DATA_BLOCK "DB59_USV_ModTCP_RCV"
{ S7_Optimized_Access := 'FALSE' }
VERSION : 0.1
NON_RETAIN
   STRUCT
      Data : Array[0..255] of Byte;
   END_STRUCT;


BEGIN

END_DATA_BLOCK

DATA_BLOCK "DB60_USV_ModTCP_SEND"
{ S7_Optimized_Access := 'FALSE' }
VERSION : 0.1
NON_RETAIN
   STRUCT
      Data : Array[0..31] of Byte;
   END_STRUCT;


BEGIN

END_DATA_BLOCK

DATA_BLOCK "DB61_USV_ModTCP_WorkData"
{ S7_Optimized_Access := 'FALSE' }
VERSION : 0.1
   STRUCT
      REQCNT : Int;
      REQ : Array[1..10] of "T_MODBUSTCP_USV_REQ";
      REQ01 : Struct   // binär
         Reg000_l : Word;   // System - UPSStatus_BF
         Reg000_h : Word;   // System - UPSStatus_BF
         Reg002 : Int;   // System - UPSStatusChangeCause_EN
         Reg003 : DWord;   // System - MOG.OutletStatus_BF
         Reg005 : Int;   // System - Reserved []
         Reg006 : DWord;   // System - SOG[0].OutletStatus_BF
         Reg008 : Int;   // System - Reserved []
         Reg009 : DWord;   // System - SOG[1].OutletStatus_BF
         Reg011 : Int;   // System - Reserved []
         Reg012 : DWord;   // System - SOG[2].OutletStatus_BF [Bitfeld]
         Reg014 : Int;   // System - Reserved []
         Reg015 : Int;   // System - Reserved []
         Reg016 : Int;   // System - Reserved []
         Reg017 : Int;   // System - Reserved []
         Reg018 : Word;   // System - SimpleSignalingStatus_BF
         Reg019 : Word;   // System - GeneralError_BF
         Reg020 : DWord;   // System - PowerSystemError_BF [Bitfeld]
         Reg022 : Word;   // System - BatterySystemError_BF
         Reg023 : Word;   // System - ReplaceBatteryTestStatus_BF
         Reg024 : Word;   // System - RunTimeCalibrationStatus_BF
         Reg025 : Word;   // System - Battery.LifeTimeStatus_BF
         Reg026 : Word;   // System - UserInterfaceStatus_BF
      END_STRUCT;
      REQ02 : Struct   // analog
         Reg128 : DInt;   // System - RunTimeRemaining [s]
         Reg130 : Int;   // System - StateOfCharge_Pct [%]
         Reg131 : Int;   // System - Battery.Positive.VoltageDC [V]
         Reg132 : Int;   // System - Battery.Negative.VoltageDC [V]
         Reg133 : Int;   // System - Battery.Date []
         Reg134 : Int;   // System - Reserved []
         Reg135 : Int;   // System - Battery.Temperature [°C]
         Reg136 : Int;   // System - Output[0].RealPower_Pct [%]
         Reg137 : Int;   // System - Output[1].RealPower_Pct [%]
         Reg138 : Int;   // System - Output[0].ApparentPower_Pct [%]
         Reg139 : Int;   // System - Output[1].ApparentPower_Pct [%]
         Reg140 : Int;   // System - Output[0].CurrentAC [A]
         Reg141 : Int;   // System - Output[1].CurrentAC [A]
         Reg142 : Int;   // System - Output[0].VoltageAC [V]
         Reg143 : Int;   // System - Output[1].VoltageAC [V]
         Reg144 : Int;   // System - Output.Frequency [Hz]
         Reg145 : DInt;   // System - Output.Energy [Wh]
         Reg147 : Int;   // System - Bypass.InputStatus_BF [Bitfeld]
         Reg148 : Int;   // System - Bypass.VoltageAC [V]
         Reg149 : Int;   // System - Bypass.Frequency [Hz]
         Reg150 : Int;   // System - Input.InputStatus_BF [Bitfeld]
         Reg151 : Int;   // System - Input[0].VoltageAC [V]
         Reg152 : Int;   // System - Input[1].VoltageAC [V]
         Reg153 : Int;   // System - Input[2].VoltageAC [V]
         Reg154 : Int;   // System - Efficiency_EN [enum]
         Reg155 : Int;   // System - MOG.TurnOffCountdown_EN [enum]
         Reg156 : Int;   // System - MOG.TurnOnCountdown_EN [enum]
         Reg157 : DInt;   // System - MOG.StayOffCountdown_EN [enum]
         Reg159 : Int;   // System - SOG[0].TurnOffCountdown_EN [enum]
         Reg160 : Int;   // System - SOG[0].TurnOnCountdown_EN [enum]
         Reg161 : DInt;   // System - SOG[0].StayOffCountdown_EN [enum]
         Reg163 : Int;   // System - SOG[1].TurnOffCountdown_EN [enum]
         Reg164 : Int;   // System - SOG[1].TurnOnCountdown_EN [enum]
         Reg165 : DInt;   // System - SOG[1].StayOffCountdown_EN [enum]
         Reg167 : Int;   // System - SOG[2].TurnOffCountdown_EN [enum]
         Reg168 : Int;   // System - SOG[2].TurnOnCountdown_EN [enum]
         Reg169 : DInt;   // System - SOG[2].StayOffCountdown_EN [enum]
      END_STRUCT;
   END_STRUCT;


BEGIN
   REQCNT := 2;
   REQ[1].TransactID := 1;
   REQ[1].UnitID := 1;
   REQ[1].FunctionCode := 3;
   REQ[1].RegisterCount := 27;
   REQ[1].SourceDB_Num := 61;
   REQ[1].SourceDB_ByteAdr := 182;
   REQ[1].SwapBytes := TRUE;
   REQ[2].TransactID := 2;
   REQ[2].UnitID := 1;
   REQ[2].FunctionCode := 3;
   REQ[2].RegisterAdr := 128;
   REQ[2].RegisterCount := 43;
   REQ[2].SourceDB_Num := 61;
   REQ[2].SourceDB_ByteAdr := 236;

END_DATA_BLOCK

DATA_BLOCK "DB_IEC_ASDUAdr"
{ S7_Optimized_Access := 'FALSE' }
AUTHOR : SIE_GST
FAMILY : S7_IEC
NAME : P_ASDUs
VERSION : 1.6
   STRUCT
      DB_Manag { ExternalVisible := 'False'} : Struct
         Pos_of_DB { ExternalVisible := 'False'} : Byte;   // reserved for future - do not change !
         No_of_all_DBs { ExternalVisible := 'False'} : Byte;   // reserved for future - do not change !
         DB_No_Act { ExternalVisible := 'False'} : Word;   // reserved for future - do not change !
         DB_No_Prev { ExternalVisible := 'False'} : Word;   // reserved for future - do not change !
         DB_No_Next { ExternalVisible := 'False'} : Word;   // reserved for future - do not change !
         Reserved { ExternalVisible := 'False'} : Word;
      END_STRUCT;
      Info_Manag { ExternalVisible := 'False'} : Struct
         P_Byte_First_Info { ExternalVisible := 'False'} : Int;   // (Byte-) Position of first Para-Block - do not change !
         No_of_Infos { ExternalVisible := 'False'} : Int;   // 0:unspecified (DB is filled up to the end); otherwise size n of ARRAY [1..n]
         Len_Info { ExternalVisible := 'False'} : USInt;   // Difference in [byte] between two Para-Blocks - do not change !
         Len_Sort_Key { ExternalVisible := 'False'} : USInt;   // 0: without sorting; >0: Data sets are sorted ascending with x bytes
         Re_internal_usage { ExternalVisible := 'False'} : DWord;
      END_STRUCT;
      Global { ExternalVisible := 'False'} : Struct
         Glob_R1 { ExternalVisible := 'False'} : Int;
         Glob_R2 { ExternalVisible := 'False'} : Word;
      END_STRUCT;
      ASDU_Adr_Para { ExternalVisible := 'False'} : Array[0..15] of Struct
         ASDU_Address { ExternalVisible := 'False'} : DInt;   // Parameter: ASDU address
         Link_Para_DB { ExternalVisible := 'False'} : Int;   // Parameter: associated link db no / 0 -> direct (no link db available)
         Link_Para_Pos { ExternalVisible := 'False'} : Int;   // Parameter: parablock no in link db
         Error { ExternalVisible := 'False'} : Bool;   // internal
         Res_1 { ExternalVisible := 'False'} : Byte;   // internal
         Res_2 { ExternalVisible := 'False'} : DInt;   // internal
         Res_3 { ExternalVisible := 'False'} : Int;   // internal
      END_STRUCT;
   END_STRUCT;


BEGIN
   Info_Manag.P_Byte_First_Info := 24;
   Info_Manag.Len_Info := 16;
   ASDU_Adr_Para[0].ASDU_Address := DINT#25602;
   ASDU_Adr_Para[1].ASDU_Address := DINT#25860;
   ASDU_Adr_Para[2].ASDU_Address := DINT#26116;
   ASDU_Adr_Para[3].ASDU_Address := DINT#26372;
   ASDU_Adr_Para[4].ASDU_Address := DINT#26628;
   ASDU_Adr_Para[5].ASDU_Address := DINT#26884;
   ASDU_Adr_Para[6].ASDU_Address := DINT#27140;
   ASDU_Adr_Para[7].ASDU_Address := DINT#27396;
   ASDU_Adr_Para[8].ASDU_Address := DINT#27652;
   ASDU_Adr_Para[9].ASDU_Address := DINT#28164;
   ASDU_Adr_Para[10].ASDU_Address := DINT#28420;
   ASDU_Adr_Para[11].ASDU_Address := DINT#28676;
   ASDU_Adr_Para[12].ASDU_Address := DINT#28932;
   ASDU_Adr_Para[13].ASDU_Address := DINT#29188;
   ASDU_Adr_Para[14].ASDU_Address := DINT#30468;
   ASDU_Adr_Para[15].ASDU_Address := DINT#5126;

END_DATA_BLOCK

DATA_BLOCK "ZEN_MW"
{ S7_Optimized_Access := 'FALSE' }
VERSION : 0.1
NON_RETAIN
   STRUCT
      Zulauf_AR_DF_ZW : DInt;   // Zulauf - Pumpwerk "Alter Rechen" - Durchfluss - Zählwert
      BB1_DF_ZW : DInt;   // Becken 1 - Ablauf - Durchfluss - Zählwert
      BB2_DF_ZW : DInt;   // Becken 2 - Ablauf - Durchfluss - Zählwert
      Zulauf_DF_ZW : DInt;   // Zulauf - Rechen - Durchfluss - Zählwert
      BB_UeSS_DF_ZW : Real;   // Becken 1+2 - Ablauf ÜSS - Durchfluss - Zählwert
      Ablauf_DF_ZW : DInt;   // Ablauf - Durchfluss - Zählwert
      Schlamm_Besch_DF_ZW : DInt;   // Schlamm - Beschickung - Durchfluss - Zählwert
      Truebwasser_DF_ZW : DInt;   // Trübwasserpumpwerk - Durchfluss - Zählwert
      BB_Biocos_DF_ZW : DInt;   // Becken 1+2 - Schlammmenge Biocos - Zählwert
      Zulauf_AR_DF_ZW_Tag : DInt;   // Zulauf - Pumpwerk "Alter Rechen" - Durchfluss - Zählwert Tag
      BB1_DF_ZW_Tag : DInt;   // Becken 1 - Ablauf - Durchfluss - Zählwert Tag
      BB2_DF_ZW_Tag : DInt;   // Becken 2 - Ablauf - Durchfluss - Zählwert Tag
      Zulauf_DF_ZW_Tag : DInt;   // Zulauf - Rechen - Durchfluss - Zählwert Tag
      BB_UeSS_DF_ZW_Tag : Real;   // Becken 1+2 - Ablauf ÜSS - Durchfluss - Zählwert Tag
      Ablauf_DF_ZW_Tag : DInt;   // Ablauf - Durchfluss - Zählwert Tag
      Schlamm_Besch_DF_ZW_Tag : DInt;   // Schlamm - Beschickung - Durchfluss - Zählwert Tag
      Truebwasser_DF_ZW_Tag : DInt;   // Trübwasserpumpwerk - Durchfluss - Zählwert Tag
      BB_Biocos_DF_ZW_Tag : DInt;   // Becken 1+2 - Schlammmenge Biocos - Zählwert Tag
      Zulauf_AR_DF_ZW_Vortag : DInt;   // Zulauf - Pumpwerk "Alter Rechen" - Durchfluss - Zählwert Vortag
      BB1_DF_ZW_Vortag : DInt;   // Becken 1 - Ablauf - Durchfluss - Zählwert Vortag
      BB2_DF_ZW_Vortag : DInt;   // Becken 2 - Ablauf - Durchfluss - Zählwert Vortag
      Zulauf_DF_ZW_Vortag : DInt;   // Zulauf - Rechen - Durchfluss - Zählwert Vortag
      BB_UeSS_DF_ZW_Vortag : Real;   // Becken 1+2 - Ablauf ÜSS - Durchfluss - Zählwert Vortag
      Ablauf_DF_ZW_Vortag : DInt;   // Ablauf - Durchfluss - Zählwert Vortag
      Schlamm_Besch_DF_ZW_Vortag : DInt;   // Schlamm - Beschickung - Durchfluss - Zählwert Vortag
      Truebwasser_DF_ZW_Vortag : DInt;   // Trübwasserpumpwerk - Durchfluss - Zählwert Vortag
      BB_Biocos_DF_ZW_Vortag : DInt;   // Becken 1+2 - Schlammmenge Biocos - Zählwert Vortag
      ZEN_Bed_ID : DInt;   // UV BG Bedienstelle - Bediener aktuell - ID
      ZEN_ESK_Stufe_act : DInt;   // UV BG - Einschaltkaskade - aktive Schaltpriorität
      ZEN_ESK_NLZ_Stufe_req : DInt;   // UV BG - Einschaltkaskade - Nachlaufzeit max. für angeforderte Schaltpriorität
      ZEN_ESK_Stufe_req : DInt;   // UV BG - Einschaltkaskade - Anforderung Schaltpriorität
      BB_Auto_GeblW_ZZ_IW : DInt;   // Steuerung Belüftung - Automatik - Zykluszeit Gebläsetausch - Istwert
      Biocos1_Auto_A_Zt_P1_SW : DInt;   // Steuerung Biocos 1 - Automatik - Sollwert A-Phase (Rechenwert U+V) - Parametersatz 1
      Biocos1_Auto_Bel_Frg_P1_SW : DInt;   // Steuerung Biocos 1 - Automatik - Sollwert Belüftungsphase Freigabe (Rechenwert V-Verz.) - Parametersatz 1
      Biocos1_Auto_A_Zt_P2_SW : DInt;   // Steuerung Biocos 1 - Automatik - Sollwert A-Phase (Rechenwert U+V) - Parametersatz 2
      Biocos1_Auto_Bel_Frg_P2_SW : DInt;   // Steuerung Biocos 1 - Automatik - Sollwert Belüftungsphase Freigabe (Rechenwert V-Verz.) - Parametersatz 2
      ZEN_Res_DB102_144_0 : DInt;   // Reserve
      Biocos1_Auto_U_Zt_Px_IW : DInt;   // Steuerung Biocos 1 - Automatik - Sollwert U-Phase - Parameter aktiv
      Biocos1_Auto_V_Zt_Px_IW : DInt;   // Steuerung Biocos 1 - Automatik - Sollwert V-Phase - Parameter aktiv
      Biocos1_Auto_A_Zt_Px_IW : DInt;   // Steuerung Biocos 1 - Automatik - Sollwert A-Phase (Rechenwert U+V) - Parameter aktiv
      Biocos1_Auto_Bel_Vz_Px_IW : DInt;   // Steuerung Biocos 1 - Automatik - Sollwert Verzögerungszeit Belüftungsphase - Parameter aktiv
      Biocos1_Auto_Bel_Frg_Px_IW : DInt;   // Steuerung Biocos 1 - Automatik - Sollwert Belüftungsphase Freigabe (Rechenwert V-Verz.) - Parameter aktiv
      Biocos1_Auto_Bel_Int_Px_IW : DInt;   // Steuerung Biocos 1 - Automatik - Sollwert Anzahl Belüftungsintervalle - Parameter aktiv
      Biocos1_Auto_Bel_Int_Zt_Px_IW : DInt;   // Steuerung Biocos 1 - Automatik - Sollwert Belüftungsdauer (fest) pro Intervall - Parameter aktiv
      Biocos1_Auto_UeSS_Zt_Px_IW : DInt;   // Steuerung Biocos 1 - Automatik - Sollwert ÜSS-Abzug Dauer - Parameter aktiv
      Biocos1_Auto_UeSS_Df_Px_IW : Real;   // Steuerung Biocos 1 - Automatik - Sollwert ÜSS-Abzug Menge - Parameter aktiv
      Biocos1_Auto_SR1_Zt_Px_IW : DInt;   // Steuerung Biocos 1 - Automatik - Sollwert Dauer Schlammrückführung SU-Becken 1 - Parameter aktiv
      Biocos1_Auto_SR2_Zt_Px_IW : DInt;   // Steuerung Biocos 1 - Automatik - Sollwert Dauer Schlammrückführung SU-Becken 2 - Parameter aktiv
      ZEN_Res_DB102_192_0 : DInt;   // Reserve
      Biocos1_Auto_UeSS_Zyk_IW : DInt;   // Steuerung Biocos 1 - Automatik - Zyklen bis ÜSS-Abzug - Istwert
      Biocos1_Auto_U1_Zt_IW : DInt;   // Steuerung Biocos 1 - Automatik - U-Phase SU-Becken 1 - Istwert
      Biocos1_Auto_V1_Zt_IW : DInt;   // Steuerung Biocos 1 - Automatik - V-Phase SU-Becken 1 - Istwert
      Biocos1_Auto_A1_Zt_IW : DInt;   // Steuerung Biocos 1 - Automatik - A-Phase SU-Becken 1 - Istwert
      Biocos1_Auto_U2_Zt_IW : DInt;   // Steuerung Biocos 1 - Automatik - U-Phase SU-Becken 2 - Istwert
      Biocos1_Auto_V2_Zt_IW : DInt;   // Steuerung Biocos 1 - Automatik - V-Phase SU-Becken 2 - Istwert
      Biocos1_Auto_A2_Zt_IW : DInt;   // Steuerung Biocos 1 - Automatik - A-Phase SU-Becken 2 - Istwert
      Biocos1_Auto_Bel_Vz_IW : DInt;   // Steuerung Biocos 1 - Automatik - Verzögerungszeit Belüftungsphase - Istwert
      Biocos1_Auto_Bel_Frg_IW : DInt;   // Steuerung Biocos 1 - Automatik - Belüftungsphase - Istwert
      Biocos1_Auto_Bel_Int_IW : DInt;   // Steuerung Biocos 1 - Automatik - Belüftungsintervall - Istwert
      Biocos1_Auto_Bel_Int_Zt_IW : DInt;   // Steuerung Biocos 1 - Automatik - Belüftungsdauer im Intervall - Istwert
      Biocos1_Auto_UeSS_Zt_IW : DInt;   // Steuerung Biocos 1 - Automatik - ÜSS-Abzug Dauer - Istwert
      Biocos1_Auto_UeSS_Df_IW : Real;   // Steuerung Biocos 1 - Automatik - ÜSS-Abzug Menge - Istwert
      Biocos1_Auto_SR1_Zt_IW : DInt;   // Steuerung Biocos 1 - Automatik - Schlammrückführung SU-Becken 1 - Istwert
      Biocos1_Auto_SR2_Zt_IW : DInt;   // Steuerung Biocos 1 - Automatik - Schlammrückführung SU-Becken 2 - Istwert
      ZEN_Res_DB102_256_0 : DInt;   // Reserve
      Biocos2_Auto_A_Zt_P1_SW : DInt;   // Steuerung Biocos 2 - Automatik - Sollwert A-Phase (Rechenwert U+V) - Parametersatz 1
      Biocos2_Auto_Bel_Frg_P1_SW : DInt;   // Steuerung Biocos 2 - Automatik - Sollwert Belüftungsphase Freigabe (Rechenwert V-Verz.) - Parametersatz 1
      Biocos2_Auto_A_Zt_P2_SW : DInt;   // Steuerung Biocos 2 - Automatik - Sollwert A-Phase (Rechenwert U+V) - Parametersatz 2
      Biocos2_Auto_Bel_Frg_P2_SW : DInt;   // Steuerung Biocos 2 - Automatik - Sollwert Belüftungsphase Freigabe (Rechenwert V-Verz.) - Parametersatz 2
      ZEN_Res_DB102_276_0 : DInt;   // Reserve
      Biocos2_Auto_U_Zt_Px_IW : DInt;   // Steuerung Biocos 2 - Automatik - Sollwert U-Phase - Parameter aktiv
      Biocos2_Auto_V_Zt_Px_IW : DInt;   // Steuerung Biocos 2 - Automatik - Sollwert V-Phase - Parameter aktiv
      Biocos2_Auto_A_Zt_Px_IW : DInt;   // Steuerung Biocos 2 - Automatik - Sollwert A-Phase (Rechenwert U+V) - Parameter aktiv
      Biocos2_Auto_Bel_Vz_Px_IW : DInt;   // Steuerung Biocos 2 - Automatik - Sollwert Verzögerungszeit Belüftungsphase - Parameter aktiv
      Biocos2_Auto_Bel_Frg_Px_IW : DInt;   // Steuerung Biocos 2 - Automatik - Sollwert Belüftungsphase Freigabe (Rechenwert V-Verz.) - Parameter aktiv
      Biocos2_Auto_Bel_Int_Px_IW : DInt;   // Steuerung Biocos 2 - Automatik - Sollwert Anzahl Belüftungsintervalle - Parameter aktiv
      Biocos2_Auto_Bel_Int_Zt_Px_IW : DInt;   // Steuerung Biocos 2 - Automatik - Sollwert Belüftungsdauer (fest) pro Intervall - Parameter aktiv
      Biocos2_Auto_UeSS_Zt_Px_IW : DInt;   // Steuerung Biocos 2 - Automatik - Sollwert ÜSS-Abzug Dauer - Parameter aktiv
      Biocos2_Auto_UeSS_Df_Px_IW : Real;   // Steuerung Biocos 2 - Automatik - Sollwert ÜSS-Abzug Menge - Parameter aktiv
      Biocos2_Auto_SR1_Zt_Px_IW : DInt;   // Steuerung Biocos 2 - Automatik - Sollwert Dauer Schlammrückführung SU-Becken 1 - Parameter aktiv
      Biocos2_Auto_SR2_Zt_Px_IW : DInt;   // Steuerung Biocos 2 - Automatik - Sollwert Dauer Schlammrückführung SU-Becken 2 - Parameter aktiv
      ZEN_Res_DB102_324_0 : DInt;   // Reserve
      Biocos2_Auto_UeSS_Zyk_IW : DInt;   // Steuerung Biocos 2 - Automatik - Zyklen bis ÜSS-Abzug - Istwert
      Biocos2_Auto_U1_Zt_IW : DInt;   // Steuerung Biocos 2 - Automatik - U-Phase SU-Becken 1 - Istwert
      Biocos2_Auto_V1_Zt_IW : DInt;   // Steuerung Biocos 2 - Automatik - V-Phase SU-Becken 1 - Istwert
      Biocos2_Auto_A1_Zt_IW : DInt;   // Steuerung Biocos 2 - Automatik - A-Phase SU-Becken 1 - Istwert
      Biocos2_Auto_U2_Zt_IW : DInt;   // Steuerung Biocos 2 - Automatik - U-Phase SU-Becken 2 - Istwert
      Biocos2_Auto_V2_Zt_IW : DInt;   // Steuerung Biocos 2 - Automatik - V-Phase SU-Becken 2 - Istwert
      Biocos2_Auto_A2_Zt_IW : DInt;   // Steuerung Biocos 2 - Automatik - A-Phase SU-Becken 2 - Istwert
      Biocos2_Auto_Bel_Vz_IW : DInt;   // Steuerung Biocos 2 - Automatik - Verzögerungszeit Belüftungsphase - Istwert
      Biocos2_Auto_Bel_Frg_IW : DInt;   // Steuerung Biocos 2 - Automatik - Belüftungsphase - Istwert
      Biocos2_Auto_Bel_Int_IW : DInt;   // Steuerung Biocos 2 - Automatik - Belüftungsintervall - Istwert
      Biocos2_Auto_Bel_Int_Zt_IW : DInt;   // Steuerung Biocos 2 - Automatik - Belüftungsdauer im Intervall - Istwert
      Biocos2_Auto_UeSS_Zt_IW : DInt;   // Steuerung Biocos 2 - Automatik - ÜSS-Abzug Dauer - Istwert
      Biocos2_Auto_UeSS_Df_IW : Real;   // Steuerung Biocos 2 - Automatik - ÜSS-Abzug Menge - Istwert
      Biocos2_Auto_SR1_Zt_IW : DInt;   // Steuerung Biocos 2 - Automatik - Schlammrückführung SU-Becken 1 - Istwert
      Biocos2_Auto_SR2_Zt_IW : DInt;   // Steuerung Biocos 2 - Automatik - Schlammrückführung SU-Becken 2 - Istwert
      Schlamm_Besch_Auto_Menge_IW : DInt;   // Steuerung Beschickung Schlammbeete - Menge Beschickung - Istwert
      PO4_Elim_DosP_Status_DF_SW : Real;   // Steuerung PO4-Elimination - Status Dosierpumpe - Menge Fällmittel - Sollwert
      PO4_Elim_DosP_Status_DF_IW : Real;   // Steuerung PO4-Elimination - Status Dosierpumpe - Menge Fällmittel - Istwert
      PO4_Elim_DosP_Status_Dr_IW : Real;   // Steuerung PO4-Elimination - Status Dosierpumpe - Druck (ohne Luftdruck) - Istwert
      PO4_Elim_DosP_Status_DF_ZW : Real;   // Steuerung PO4-Elimination - Status Dosierpumpe - Menge Fällmittel - Zählwert
      Biocos1_Auto_Bel_O2_Reg_IW : Real;   // Steuerung Biocos 1 - Automatik O2-Regler - Vorgabe Automatik Blockdrehzahl für Ansteuerung Gebläse
      Biocos2_Auto_Bel_O2_Reg_IW : Real;   // Steuerung Biocos 2 - Automatik O2-Regler - Vorgabe Automatik Blockdrehzahl für Ansteuerung Gebläse
      BB_G1_KS_Druck_Netz : Real;   // Belebung - SigmaControl Gebläse 1 - Messwerte - Netzdruck
      BB_G1_KS_Temp_Verdicht : Real;   // Belebung - SigmaControl Gebläse 1 - Messwerte - Verdichtungsendtemperatur (t2)
      BB_G1_KS_Temp_Schallhaube : Real;   // Belebung - SigmaControl Gebläse 1 - Messwerte - Temperatur Schalldämmhaube (t_S)
      BB_G1_KS_Temp_Ansaug : Real;   // Belebung - SigmaControl Gebläse 1 - Messwerte - Ansaugtemperatur (t1)
      BB_G1_KS_Temp_Oel : Real;   // Belebung - SigmaControl Gebläse 1 - Messwerte - Öltemperatur (t3 )
      BB_G1_KS_Temp_Wicklung : Real;   // Belebung - SigmaControl Gebläse 1 - Messwerte - Wicklungstemperatur Hauptmotor
      BB_G1_KS_Volumenstrom : Real;   // Belebung - SigmaControl Gebläse 1 - Messwerte - Volumenstrom
      BB_G1_KS_Motorfrequenz : Real;   // Belebung - SigmaControl Gebläse 1 - Messwerte - Motorfrequenz
      BB_G1_KS_Motordrehzahl : Real;   // Belebung - SigmaControl Gebläse 1 - Messwerte - Motordrehzahl
      BB_G1_KS_Blockdrehzahl : Real;   // Belebung - SigmaControl Gebläse 1 - Messwerte - Blockdrehzahl
      BB_G2_KS_Druck_Netz : Real;   // Belebung - SigmaControl Gebläse 2 - Messwerte - Netzdruck
      BB_G2_KS_Temp_Verdicht : Real;   // Belebung - SigmaControl Gebläse 2 - Messwerte - Verdichtungsendtemperatur (t2)
      BB_G2_KS_Temp_Schallhaube : Real;   // Belebung - SigmaControl Gebläse 2 - Messwerte - Temperatur Schalldämmhaube (t_S)
      BB_G2_KS_Temp_Ansaug : Real;   // Belebung - SigmaControl Gebläse 2 - Messwerte - Ansaugtemperatur (t1)
      BB_G2_KS_Temp_Oel : Real;   // Belebung - SigmaControl Gebläse 2 - Messwerte - Öltemperatur (t3 )
      BB_G2_KS_Temp_Wicklung : Real;   // Belebung - SigmaControl Gebläse 2 - Messwerte - Wicklungstemperatur Hauptmotor
      BB_G2_KS_Volumenstrom : Real;   // Belebung - SigmaControl Gebläse 2 - Messwerte - Volumenstrom
      BB_G2_KS_Motorfrequenz : Real;   // Belebung - SigmaControl Gebläse 2 - Messwerte - Motorfrequenz
      BB_G2_KS_Motordrehzahl : Real;   // Belebung - SigmaControl Gebläse 2 - Messwerte - Motordrehzahl
      BB_G2_KS_Blockdrehzahl : Real;   // Belebung - SigmaControl Gebläse 2 - Messwerte - Blockdrehzahl
      BB_G3_KS_Druck_Netz : Real;   // Belebung - SigmaControl Gebläse 3 - Messwerte - Netzdruck
      BB_G3_KS_Temp_Verdicht : Real;   // Belebung - SigmaControl Gebläse 3 - Messwerte - Verdichtungsendtemperatur (t2)
      BB_G3_KS_Temp_Schallhaube : Real;   // Belebung - SigmaControl Gebläse 3 - Messwerte - Temperatur Schalldämmhaube (t_S)
      BB_G3_KS_Temp_Ansaug : Real;   // Belebung - SigmaControl Gebläse 3 - Messwerte - Ansaugtemperatur (t1)
      BB_G3_KS_Temp_Oel : Real;   // Belebung - SigmaControl Gebläse 3 - Messwerte - Öltemperatur (t3 )
      BB_G3_KS_Temp_Wicklung : Real;   // Belebung - SigmaControl Gebläse 3 - Messwerte - Wicklungstemperatur Hauptmotor
      BB_G3_KS_Volumenstrom : Real;   // Belebung - SigmaControl Gebläse 3 - Messwerte - Volumenstrom
      BB_G3_KS_Motorfrequenz : Real;   // Belebung - SigmaControl Gebläse 3 - Messwerte - Motorfrequenz
      BB_G3_KS_Motordrehzahl : Real;   // Belebung - SigmaControl Gebläse 3 - Messwerte - Motordrehzahl
      BB_G3_KS_Blockdrehzahl : Real;   // Belebung - SigmaControl Gebläse 3 - Messwerte - Blockdrehzahl
      Umwelt_RM_ZW : Real;   // Wetterstation - Regenmenge - Zählwert
      Umwelt_RM_ZW_Tag : Real;   // Wetterstation - Regenmenge - Zählwert Tag
      Umwelt_RM_ZW_Vortag : Real;   // Wetterstation - Regenmenge - Zählwert Vortag
      RunTimeRemaining : Real;   // USV-Anlage - Status - verbleibende Laufzeit
      StateOfCharge_Pct : Real;   // USV-Anlage - Status - Batterieladung
      RES : Array[0..9] of Byte;
   END_STRUCT;


BEGIN
   Zulauf_AR_DF_ZW := 583302;
   BB1_DF_ZW := 0;
   BB2_DF_ZW := 0;
   Zulauf_DF_ZW := 1741318;
   BB_UeSS_DF_ZW := 82177.4;
   Ablauf_DF_ZW := 1542271;
   Schlamm_Besch_DF_ZW := 53300;
   Truebwasser_DF_ZW := 207644;
   BB_Biocos_DF_ZW := 0;
   Zulauf_AR_DF_ZW_Tag := 0;
   BB1_DF_ZW_Tag := 0;
   BB2_DF_ZW_Tag := 0;
   Zulauf_DF_ZW_Tag := 1066;
   BB_UeSS_DF_ZW_Tag := 39.0;
   Ablauf_DF_ZW_Tag := 869;
   Schlamm_Besch_DF_ZW_Tag := 0;
   Truebwasser_DF_ZW_Tag := 89;
   BB_Biocos_DF_ZW_Tag := 0;
   Zulauf_AR_DF_ZW_Vortag := 0;
   BB1_DF_ZW_Vortag := 0;
   BB2_DF_ZW_Vortag := 0;
   Zulauf_DF_ZW_Vortag := 905;
   BB_UeSS_DF_ZW_Vortag := 39.0;
   Ablauf_DF_ZW_Vortag := 815;
   Schlamm_Besch_DF_ZW_Vortag := 0;
   Truebwasser_DF_ZW_Vortag := 90;
   BB_Biocos_DF_ZW_Vortag := 0;
   ZEN_Bed_ID := 0;
   ZEN_ESK_Stufe_act := 0;
   ZEN_ESK_NLZ_Stufe_req := 0;
   ZEN_ESK_Stufe_req := 0;
   BB_Auto_GeblW_ZZ_IW := 22;
   Biocos1_Auto_A_Zt_P1_SW := 60;
   Biocos1_Auto_Bel_Frg_P1_SW := 33;
   Biocos1_Auto_A_Zt_P2_SW := 90;
   Biocos1_Auto_Bel_Frg_P2_SW := 71;
   ZEN_Res_DB102_144_0 := 0;
   Biocos1_Auto_U_Zt_Px_IW := 15;
   Biocos1_Auto_V_Zt_Px_IW := 45;
   Biocos1_Auto_A_Zt_Px_IW := 60;
   Biocos1_Auto_Bel_Vz_Px_IW := 720;
   Biocos1_Auto_Bel_Frg_Px_IW := 33;
   Biocos1_Auto_Bel_Int_Px_IW := 3;
   Biocos1_Auto_Bel_Int_Zt_Px_IW := 300;
   Biocos1_Auto_UeSS_Zt_Px_IW := 8;
   Biocos1_Auto_UeSS_Df_Px_IW := 1.6;
   Biocos1_Auto_SR1_Zt_Px_IW := 3;
   Biocos1_Auto_SR2_Zt_Px_IW := 3;
   ZEN_Res_DB102_192_0 := 0;
   Biocos1_Auto_UeSS_Zyk_IW := 1;
   Biocos1_Auto_U1_Zt_IW := 15;
   Biocos1_Auto_V1_Zt_IW := 45;
   Biocos1_Auto_A1_Zt_IW := 4;
   Biocos1_Auto_U2_Zt_IW := 15;
   Biocos1_Auto_V2_Zt_IW := 4;
   Biocos1_Auto_A2_Zt_IW := 60;
   Biocos1_Auto_Bel_Vz_IW := 720;
   Biocos1_Auto_Bel_Frg_IW := 4;
   Biocos1_Auto_Bel_Int_IW := 0;
   Biocos1_Auto_Bel_Int_Zt_IW := 183;
   Biocos1_Auto_UeSS_Zt_IW := 8;
   Biocos1_Auto_UeSS_Df_IW := 1.695313;
   Biocos1_Auto_SR1_Zt_IW := 3;
   Biocos1_Auto_SR2_Zt_IW := 3;
   ZEN_Res_DB102_256_0 := 0;
   Biocos2_Auto_A_Zt_P1_SW := 60;
   Biocos2_Auto_Bel_Frg_P1_SW := 33;
   Biocos2_Auto_A_Zt_P2_SW := 90;
   Biocos2_Auto_Bel_Frg_P2_SW := 71;
   ZEN_Res_DB102_276_0 := 0;
   Biocos2_Auto_U_Zt_Px_IW := 15;
   Biocos2_Auto_V_Zt_Px_IW := 45;
   Biocos2_Auto_A_Zt_Px_IW := 60;
   Biocos2_Auto_Bel_Vz_Px_IW := 720;
   Biocos2_Auto_Bel_Frg_Px_IW := 33;
   Biocos2_Auto_Bel_Int_Px_IW := 3;
   Biocos2_Auto_Bel_Int_Zt_Px_IW := 300;
   Biocos2_Auto_UeSS_Zt_Px_IW := 8;
   Biocos2_Auto_UeSS_Df_Px_IW := 1.6;
   Biocos2_Auto_SR1_Zt_Px_IW := 3;
   Biocos2_Auto_SR2_Zt_Px_IW := 3;
   ZEN_Res_DB102_324_0 := 0;
   Biocos2_Auto_UeSS_Zyk_IW := 0;
   Biocos2_Auto_U1_Zt_IW := 15;
   Biocos2_Auto_V1_Zt_IW := 4;
   Biocos2_Auto_A1_Zt_IW := 60;
   Biocos2_Auto_U2_Zt_IW := 15;
   Biocos2_Auto_V2_Zt_IW := 45;
   Biocos2_Auto_A2_Zt_IW := 4;
   Biocos2_Auto_Bel_Vz_IW := 720;
   Biocos2_Auto_Bel_Frg_IW := 4;
   Biocos2_Auto_Bel_Int_IW := 0;
   Biocos2_Auto_Bel_Int_Zt_IW := 217;
   Biocos2_Auto_UeSS_Zt_IW := 8;
   Biocos2_Auto_UeSS_Df_IW := 1.601563;
   Biocos2_Auto_SR1_Zt_IW := 3;
   Biocos2_Auto_SR2_Zt_IW := 3;
   Schlamm_Besch_Auto_Menge_IW := 50;
   PO4_Elim_DosP_Status_DF_SW := 0.2077;
   PO4_Elim_DosP_Status_DF_IW := 0.2053;
   PO4_Elim_DosP_Status_Dr_IW := 1.0;
   PO4_Elim_DosP_Status_DF_ZW := 34901.2;
   Biocos1_Auto_Bel_O2_Reg_IW := 3000.0;
   Biocos2_Auto_Bel_O2_Reg_IW := 3000.0;
   BB_G1_KS_Druck_Netz := 576.0;
   BB_G1_KS_Temp_Verdicht := 63.9;
   BB_G1_KS_Temp_Schallhaube := -3276.8;
   BB_G1_KS_Temp_Ansaug := 20.7;
   BB_G1_KS_Temp_Oel := 37.5;
   BB_G1_KS_Temp_Wicklung := 45.6;
   BB_G1_KS_Volumenstrom := 294.0;
   BB_G1_KS_Motorfrequenz := 17.0;
   BB_G1_KS_Motordrehzahl := 1055.0;
   BB_G1_KS_Blockdrehzahl := 2997.0;
   BB_G2_KS_Druck_Netz := 565.0;
   BB_G2_KS_Temp_Verdicht := 63.9;
   BB_G2_KS_Temp_Schallhaube := -3276.8;
   BB_G2_KS_Temp_Ansaug := 20.7;
   BB_G2_KS_Temp_Oel := 35.5;
   BB_G2_KS_Temp_Wicklung := 44.1;
   BB_G2_KS_Volumenstrom := 300.0;
   BB_G2_KS_Motorfrequenz := 17.0;
   BB_G2_KS_Motordrehzahl := 1057.0;
   BB_G2_KS_Blockdrehzahl := 3003.0;
   BB_G3_KS_Druck_Netz := 0.0;
   BB_G3_KS_Temp_Verdicht := 18.8;
   BB_G3_KS_Temp_Schallhaube := -3276.8;
   BB_G3_KS_Temp_Ansaug := 18.6;
   BB_G3_KS_Temp_Oel := 18.7;
   BB_G3_KS_Temp_Wicklung := 18.3;
   BB_G3_KS_Volumenstrom := 0.0;
   BB_G3_KS_Motorfrequenz := 0.0;
   BB_G3_KS_Motordrehzahl := 0.0;
   BB_G3_KS_Blockdrehzahl := 0.0;
   RES[0] := 16#00;
   RES[1] := 16#00;
   RES[2] := 16#00;
   RES[3] := 16#00;
   RES[4] := 16#00;
   RES[5] := 16#00;
   RES[6] := 16#00;
   RES[7] := 16#00;
   RES[8] := 16#00;
   RES[9] := 16#00;

END_DATA_BLOCK

DATA_BLOCK "ZEN_Meld"
{ S7_Optimized_Access := 'FALSE' }
VERSION : 0.1
   STRUCT
      E_Zulauf_AR_P1_Ein : Bool;   // Zulauf - Pumpwerk "Alter Rechen" - Pumpe 1 - Betrieb
      E_Zulauf_AR_P1_St : Bool;   // Zulauf - Pumpwerk "Alter Rechen" - Pumpe 1 - Störung
      E_Zulauf_AR_SS : Bool;   // Zulauf - Pumpwerk "Alter Rechen" - Sammelstörung
      E_Zulauf_AR_P2_Ein : Bool;   // Zulauf - Pumpwerk "Alter Rechen" - Pumpe 2 - Betrieb
      E_Zulauf_AR_P2_St : Bool;   // Zulauf - Pumpwerk "Alter Rechen" - Pumpe 2 - Störung
      E_Zulauf_AR_HW : Bool;   // Zulauf - Pumpwerk "Alter Rechen" - Hochwasser
      E_Zulauf_AR_Niv_St : Bool;   // Zulauf - Pumpwerk "Alter Rechen" - Niveau - Störung
      E_Zulauf_AR_DF_ZI : Bool;   // Zulauf - Pumpwerk "Alter Rechen" - Durchfluss - Impuls
      E_Zulauf_AR_DF_St : Bool;   // Zulauf - Pumpwerk "Alter Rechen" - Durchfluss - Störung
      E_Ablauf_pH_St : Bool;   // Ablauf - pH-Wert - Störung
      E_Ablauf_O2_St : Bool;   // Ablauf - O2-Gehalt - Störung
      E_Ablauf_DF_ZI : Bool;   // Ablauf - Durchfluss - Impuls
      E_Ablauf_DF_St : Bool;   // Ablauf - Durchfluss - Störung
      E_BB_UeSS_DF_ZI : Bool;   // Becken 1+2 - Ablauf ÜSS - Durchfluss - Impuls
      E_ZEN_Res_1_6 : Bool;   // Reserve
      E_ZEN_Res_1_7 : Bool;   // Reserve
      E_NSHV_SS1_St : Bool;   // NSHV Steuerspannungsüberwachung 1 - Störung
      E_NSHV_SS2_St : Bool;   // NSHV Steuerspannungsüberwachung 2 - Störung
      E_NSHV_N02_AF_St : Bool;   // NSHV Sicherungsüberwachung Feld N02 - Störung
      E_NSHV_N03_AF_St : Bool;   // NSHV Sicherungsüberwachung Feld N03 - Störung
      E_NSHV_N04_AF_St : Bool;   // NSHV Sicherungsüberwachung Feld N04 - Störung
      E_NSHV_LS_Aus : Bool;   // NSHV Netzleistungsschalter - Aus
      E_NSHV_LS_St : Bool;   // NSHV Netzleistungsschalter - ausgelöst
      E_NSHV_NA : Bool;   // NSHV Netzspannungsüberwachung - ausgelöst
      E_ZEN_Res_3_0 : Bool;   // Reserve
      E_ZEN_Res_3_1 : Bool;   // Reserve
      E_ZEN_Res_3_2 : Bool;   // Reserve
      E_ZEN_Res_3_3 : Bool;   // Reserve
      E_ZEN_Res_3_4 : Bool;   // Reserve
      E_ZEN_Res_3_5 : Bool;   // Reserve
      E_ZEN_Res_3_6 : Bool;   // Reserve
      E_ZEN_Res_3_7 : Bool;   // Reserve
      E_BB_G1_Ein : Bool;   // Belebung - Gebläse 1 - Betrieb
      E_BB_G1_St : Bool;   // Belebung - Gebläse 1 - Störung
      E_BB_G1_Bed_vOrt : Bool;   // Belebung - Gebläse 1 - vor-Ort-Hand
      E_BB_G1_Bed_Fern : Bool;   // Belebung - Gebläse 1 - vor-Ort-Fern
      E_BB_G1_AF_St : Bool;   // Belebung - Gebläse 1 - Steuersicherung ausgelöst
      E_BB_SHL_G1_Ein : Bool;   // Belebung - Schallhaubenlüfter Gebläse 1 - Betrieb
      E_BB_SHL_G1_St : Bool;   // Belebung - Schallhaubenlüfter Gebläse 1 - Störung
      E_BB_G2_Ein : Bool;   // Belebung - Gebläse 2 - Betrieb
      E_BB_G2_St : Bool;   // Belebung - Gebläse 2 - Störung
      E_BB_G2_Bed_vOrt : Bool;   // Belebung - Gebläse 2 - vor-Ort-Hand
      E_BB_G2_Bed_Fern : Bool;   // Belebung - Gebläse 2 - vor-Ort-Fern
      E_BB_G2_AF_St : Bool;   // Belebung - Gebläse 2 - Steuersicherung ausgelöst
      E_BB_SHL_G2_Ein : Bool;   // Belebung - Schallhaubenlüfter Gebläse 2 - Betrieb
      E_BB_SHL_G2_St : Bool;   // Belebung - Schallhaubenlüfter Gebläse 2 - Störung
      E_BB_G3_Ein : Bool;   // Belebung - Gebläse 3 - Betrieb
      E_BB_G3_St : Bool;   // Belebung - Gebläse 3 - Störung
      E_BB_G3_Bed_vOrt : Bool;   // Belebung - Gebläse 3 - vor-Ort-Hand
      E_BB_G3_Bed_Fern : Bool;   // Belebung - Gebläse 3 - vor-Ort-Fern
      E_BB_G3_AF_St : Bool;   // Belebung - Gebläse 3 - Steuersicherung ausgelöst
      E_BB_SHL_G3_Ein : Bool;   // Belebung - Schallhaubenlüfter Gebläse 3 - Betrieb
      E_BB_SHL_G3_St : Bool;   // Belebung - Schallhaubenlüfter Gebläse 3 - Störung
      E_BB_AV_Ein : Bool;   // Belebung - Gebläsestation - Abluftventilator - Betrieb
      E_BB_AV_St : Bool;   // Belebung - Gebläsestation - Abluftventilator - Störung
      E_BB_AV_AF_St : Bool;   // Belebung - Gebläsestation - Abluftventilator - Steuersicherung ausgelöst
      E_BB_RT : Bool;   // Belebung - Gebläsestation - Raumthermostat - Grenztemperatur erreicht
      E_BB1_SR_K_Ein : Bool;   // Becken 1 - Druckluftkompressor Schlammrückführung
      E_BB1_SR_K_St : Bool;   // Becken 1 - Druckluftkompressor Schlammrückführung
      E_BB1_SR_K_AF_St : Bool;   // Becken 1 - Druckluftkompressor Schlammrückführung
      E_BB_LS1_EA : Bool;   // Belebung - Gebläsestation - Luftwegschieber 1 - Endlage Auf
      E_BB_LS1_EZ : Bool;   // Belebung - Gebläsestation - Luftwegschieber 1 - Endlage Zu
      E_BB_LS1_St : Bool;   // Belebung - Gebläsestation - Luftwegschieber 1 - Störung
      E_BB_LS1_Bed_vOrt : Bool;   // Belebung - Gebläsestation - Luftwegschieber 1 - vor-Ort-Hand
      E_BB_LS1_Bed_Fern : Bool;   // Belebung - Gebläsestation - Luftwegschieber 1 - vor-Ort-Fern
      E_BB_LS1_AF_St : Bool;   // Belebung - Gebläsestation - Luftwegschieber 1 - Steuersicherung ausgelöst
      E_BB_LS2_EA : Bool;   // Belebung - Gebläsestation - Luftwegschieber 2 - Endlage Auf
      E_BB_LS2_EZ : Bool;   // Belebung - Gebläsestation - Luftwegschieber 2 - Endlage Zu
      E_BB_LS2_St : Bool;   // Belebung - Gebläsestation - Luftwegschieber 2 - Störung
      E_BB_LS2_Bed_vOrt : Bool;   // Belebung - Gebläsestation - Luftwegschieber 2 - vor-Ort-Hand
      E_BB_LS2_Bed_Fern : Bool;   // Belebung - Gebläsestation - Luftwegschieber 2 - vor-Ort-Fern
      E_BB_LS2_AF_St : Bool;   // Belebung - Gebläsestation - Luftwegschieber 2 - Steuersicherung ausgelöst
      E_BB1_RZP1_Ein : Bool;   // Becken 1 - Rezipumpe 1 - Betrieb
      E_BB1_RZP1_St : Bool;   // Becken 1 - Rezipumpe 1 - Störung
      E_BB1_RZP1_Bed_vOrt : Bool;   // Becken 1 - Rezipumpe 1 - vor-Ort-Hand
      E_BB1_RZP1_Bed_Fern : Bool;   // Becken 1 - Rezipumpe 1 - vor-Ort-Fern
      E_BB1_RZP1_AF_St : Bool;   // Becken 1 - Rezipumpe 1 - Steuersicherung ausgelöst
      E_BB1_RZP2_Ein : Bool;   // Becken 1 - Rezipumpe 2 - Betrieb
      E_BB1_RZP2_St : Bool;   // Becken 1 - Rezipumpe 2 - Störung
      E_BB1_RZP2_Bed_vOrt : Bool;   // Becken 1 - Rezipumpe 2 - vor-Ort-Hand
      E_BB1_RZP2_Bed_Fern : Bool;   // Becken 1 - Rezipumpe 2 - vor-Ort-Fern
      E_BB1_RZP2_AF_St : Bool;   // Becken 1 - Rezipumpe 2 - Steuersicherung ausgelöst
      E_BB1_UeSP_Ein : Bool;   // Becken 1 - ÜSS-Pumpe - Betrieb
      E_BB1_UeSP_St : Bool;   // Becken 1 - ÜSS-Pumpe - Störung
      E_BB1_UeSP_Bed_vOrt : Bool;   // Becken 1 - ÜSS-Pumpe - vor-Ort-Hand
      E_BB1_UeSP_Bed_Fern : Bool;   // Becken 1 - ÜSS-Pumpe - vor-Ort-Fern
      E_BB1_UeSP_AF_St : Bool;   // Becken 1 - ÜSS-Pumpe - Steuersicherung ausgelöst
      E_BB1_AS1_EA : Bool;   // Becken 1 - Ablaufschieber 1 - Endlage Auf
      E_BB1_AS1_EZ : Bool;   // Becken 1 - Ablaufschieber 1 - Endlage Zu
      E_BB1_AS1_St : Bool;   // Becken 1 - Ablaufschieber 1 - Störung
      E_BB1_AS1_Bed_vOrt : Bool;   // Becken 1 - Ablaufschieber 1 - vor-Ort-Hand
      E_BB1_AS1_Bed_Fern : Bool;   // Becken 1 - Ablaufschieber 1 - vor-Ort-Fern
      E_BB1_AS1_AF_St : Bool;   // Becken 1 - Ablaufschieber 1 - Steuersicherung ausgelöst
      E_BB1_AS2_EA : Bool;   // Becken 1 - Ablaufschieber 2 - Endlage Auf
      E_BB1_AS2_EZ : Bool;   // Becken 1 - Ablaufschieber 2 - Endlage Zu
      E_BB1_AS2_St : Bool;   // Becken 1 - Ablaufschieber 2 - Störung
      E_BB1_AS2_Bed_vOrt : Bool;   // Becken 1 - Ablaufschieber 2 - vor-Ort-Hand
      E_BB1_AS2_Bed_Fern : Bool;   // Becken 1 - Ablaufschieber 2 - vor-Ort-Fern
      E_BB1_AS2_AF_St : Bool;   // Becken 1 - Ablaufschieber 2 - Steuersicherung ausgelöst
      E_BB1_SR1_Anst : Bool;   // Becken 1 - MV Schlammrückführung 1 - Ansteuerung
      E_BB1_SR1_Bed_vOrt : Bool;   // Becken 1 - MV Schlammrückführung 1 - vor-Ort-Hand
      E_BB1_SR1_Bed_Fern : Bool;   // Becken 1 - MV Schlammrückführung 1 - vor-Ort-Fern
      E_BB1_SR1_AF_St : Bool;   // Becken 1 - MV Schlammrückführung 1 - Steuersicherung ausgelöst
      E_BB1_SR2_Anst : Bool;   // Becken 1 - MV Schlammrückführung 2 - Ansteuerung
      E_BB1_SR2_Bed_vOrt : Bool;   // Becken 1 - MV Schlammrückführung 2 - vor-Ort-Hand
      E_BB1_SR2_Bed_Fern : Bool;   // Becken 1 - MV Schlammrückführung 2 - vor-Ort-Fern
      E_BB1_SR2_AF_St : Bool;   // Becken 1 - MV Schlammrückführung 2 - Steuersicherung ausgelöst
      E_BB1_O2_St : Bool;   // Becken 1 - O2-Gehalt - Störung
      E_BB1_DF_ZI : Bool;   // Becken 1 - Ablauf - Durchfluss - Impuls
      E_BB1_DF_St : Bool;   // Becken 1 - Ablauf - Durchfluss - Störung
      E_BB2_RZP1_Ein : Bool;   // Becken 2 - Rezipumpe 1 - Betrieb
      E_BB2_RZP1_St : Bool;   // Becken 2 - Rezipumpe 1 - Störung
      E_BB2_RZP1_Bed_vOrt : Bool;   // Becken 2 - Rezipumpe 1 - vor-Ort-Hand
      E_BB2_RZP1_Bed_Fern : Bool;   // Becken 2 - Rezipumpe 1 - vor-Ort-Fern
      E_BB2_RZP1_AF_St : Bool;   // Becken 2 - Rezipumpe 1 - Steuersicherung ausgelöst
      E_BB2_RZP2_Ein : Bool;   // Becken 2 - Rezipumpe 2 - Betrieb
      E_BB2_RZP2_St : Bool;   // Becken 2 - Rezipumpe 2 - Störung
      E_BB2_RZP2_Bed_vOrt : Bool;   // Becken 2 - Rezipumpe 2 - vor-Ort-Hand
      E_BB2_RZP2_Bed_Fern : Bool;   // Becken 2 - Rezipumpe 2 - vor-Ort-Fern
      E_BB2_RZP2_AF_St : Bool;   // Becken 2 - Rezipumpe 2 - Steuersicherung ausgelöst
      E_BB2_UeSP_Ein : Bool;   // Becken 2 - ÜSS-Pumpe - Betrieb
      E_BB2_UeSP_St : Bool;   // Becken 2 - ÜSS-Pumpe - Störung
      E_BB2_UeSP_Bed_vOrt : Bool;   // Becken 2 - ÜSS-Pumpe - vor-Ort-Hand
      E_BB2_UeSP_Bed_Fern : Bool;   // Becken 2 - ÜSS-Pumpe - vor-Ort-Fern
      E_BB2_UeSP_AF_St : Bool;   // Becken 2 - ÜSS-Pumpe - Steuersicherung ausgelöst
      E_BB2_AS1_EA : Bool;   // Becken 2 - Ablaufschieber 1 - Endlage Auf
      E_BB2_AS1_EZ : Bool;   // Becken 2 - Ablaufschieber 1 - Endlage Zu
      E_BB2_AS1_St : Bool;   // Becken 2 - Ablaufschieber 1 - Störung
      E_BB2_AS1_Bed_vOrt : Bool;   // Becken 2 - Ablaufschieber 1 - vor-Ort-Hand
      E_BB2_AS1_Bed_Fern : Bool;   // Becken 2 - Ablaufschieber 1 - vor-Ort-Fern
      E_BB2_AS1_AF_St : Bool;   // Becken 2 - Ablaufschieber 1 - Steuersicherung ausgelöst
      E_BB2_AS2_EA : Bool;   // Becken 2 - Ablaufschieber 2 - Endlage Auf
      E_BB2_AS2_EZ : Bool;   // Becken 2 - Ablaufschieber 2 - Endlage Zu
      E_BB2_AS2_St : Bool;   // Becken 2 - Ablaufschieber 2 - Störung
      E_BB2_AS2_Bed_vOrt : Bool;   // Becken 2 - Ablaufschieber 2 - vor-Ort-Hand
      E_BB2_AS2_Bed_Fern : Bool;   // Becken 2 - Ablaufschieber 2 - vor-Ort-Fern
      E_BB2_AS2_AF_St : Bool;   // Becken 2 - Ablaufschieber 2 - Steuersicherung ausgelöst
      E_BB2_SR1_Anst : Bool;   // Becken 2 - MV Schlammrückführung 1 - Ansteuerung
      E_BB2_SR1_Bed_vOrt : Bool;   // Becken 2 - MV Schlammrückführung 1 - vor-Ort-Hand
      E_BB2_SR1_Bed_Fern : Bool;   // Becken 2 - MV Schlammrückführung 1 - vor-Ort-Fern
      E_BB2_SR1_AF_St : Bool;   // Becken 2 - MV Schlammrückführung 1 - Steuersicherung ausgelöst
      E_BB2_SR2_Anst : Bool;   // Becken 2 - MV Schlammrückführung 2 - Ansteuerung
      E_BB2_SR2_Bed_vOrt : Bool;   // Becken 2 - MV Schlammrückführung 2 - vor-Ort-Hand
      E_BB2_SR2_Bed_Fern : Bool;   // Becken 2 - MV Schlammrückführung 2 - vor-Ort-Fern
      E_BB2_SR2_AF_St : Bool;   // Becken 2 - MV Schlammrückführung 2 - Steuersicherung ausgelöst
      E_BB2_O2_St : Bool;   // Becken 2 - O2-Gehalt - Störung
      E_BB2_DF_ZI : Bool;   // Becken 2 - Ablauf - Durchfluss - Impuls
      E_BB2_DF_St : Bool;   // Becken 2 - Ablauf - Durchfluss - Störung
      E_BB2_SR_K_Ein : Bool;   // Becken 2 - Druckluftkompressor Schlammrückführung
      E_BB2_SR_K_St : Bool;   // Becken 2 - Druckluftkompressor Schlammrückführung
      E_BB2_SR_K_AF_St : Bool;   // Becken 2 - Druckluftkompressor Schlammrückführung
      E_ZEN_Res_26_7 : Bool;   // Reserve
      E_ZEN_Res_27_0 : Bool;   // Reserve
      E_ZEN_Res_27_1 : Bool;   // Reserve
      E_ZEN_Res_27_2 : Bool;   // Reserve
      E_ZEN_Res_27_3 : Bool;   // Reserve
      E_ZEN_Res_27_4 : Bool;   // Reserve
      E_ZEN_Res_27_5 : Bool;   // Reserve
      E_ZEN_Res_27_6 : Bool;   // Reserve
      E_ZEN_Res_27_7 : Bool;   // Reserve
      A_BB_G1_Ein : Bool;   // Belebung - Gebläse 1 - Ansteuerung Ein
      A_BB_G2_Ein : Bool;   // Belebung - Gebläse 2 - Ansteuerung Ein
      A_BB_G3_Ein : Bool;   // Belebung - Gebläse 3 - Ansteuerung Ein
      A_BB_LS1_Auf : Bool;   // Belebung - Gebläsestation - Luftwegschieber 1 - Ansteuerung Auf
      A_BB_LS1_Zu : Bool;   // Belebung - Gebläsestation - Luftwegschieber 1 - Ansteuerung Zu
      A_BB_LS2_Auf : Bool;   // Belebung - Gebläsestation - Luftwegschieber 2 - Ansteuerung Auf
      A_BB_LS2_Zu : Bool;   // Belebung - Gebläsestation - Luftwegschieber 2 - Ansteuerung Zu
      A_ZEN_Res_12_7 : Bool;   // Reserve
      A_BB1_RZP1_Ein : Bool;   // Becken 1 - Rezipumpe 1 - Ansteuerung Ein
      A_BB1_RZP2_Ein : Bool;   // Becken 1 - Rezipumpe 2 - Ansteuerung Ein
      A_BB1_UeSP_Ein : Bool;   // Becken 1 - ÜSS-Pumpe - Ansteuerung Ein
      A_BB1_AS1_Auf : Bool;   // Becken 1 - Ablaufschieber 1 - Ansteuerung Auf
      A_BB1_AS1_Zu : Bool;   // Becken 1 - Ablaufschieber 1 - Ansteuerung Zu
      A_BB1_AS2_Auf : Bool;   // Becken 1 - Ablaufschieber 2 - Ansteuerung Auf
      A_BB1_AS2_Zu : Bool;   // Becken 1 - Ablaufschieber 2 - Ansteuerung Zu
      A_BB1_SR1_Auf : Bool;   // Becken 1 - MV Schlammrückführung 1 - Ansteuerung Auf
      A_BB1_SR2_Auf : Bool;   // Becken 1 - MV Schlammrückführung 2 - Ansteuerung Auf
      A_ZEN_Res_14_1 : Bool;   // Reserve
      A_ZEN_Res_14_2 : Bool;   // Reserve
      A_ZEN_Res_14_3 : Bool;   // Reserve
      A_ZEN_Res_14_4 : Bool;   // Reserve
      A_ZEN_Res_14_5 : Bool;   // Reserve
      A_ZEN_Res_14_6 : Bool;   // Reserve
      A_ZEN_Res_14_7 : Bool;   // Reserve
      A_BB2_RZP1_Ein : Bool;   // Becken 2 - Rezipumpe 1 - Ansteuerung Ein
      A_BB2_RZP2_Ein : Bool;   // Becken 2 - Rezipumpe 2 - Ansteuerung Ein
      A_BB2_UeSP_Ein : Bool;   // Becken 2 - ÜSS-Pumpe - Ansteuerung Ein
      A_BB2_AS1_Auf : Bool;   // Becken 2 - Ablaufschieber 1 - Ansteuerung Auf
      A_BB2_AS1_Zu : Bool;   // Becken 2 - Ablaufschieber 1 - Ansteuerung Zu
      A_BB2_AS2_Auf : Bool;   // Becken 2 - Ablaufschieber 2 - Ansteuerung Auf
      A_BB2_AS2_Zu : Bool;   // Becken 2 - Ablaufschieber 2 - Ansteuerung Zu
      A_BB2_SR1_Auf : Bool;   // Becken 2 - MV Schlammrückführung 1 - Ansteuerung Auf
      A_BB2_SR2_Auf : Bool;   // Becken 2 - MV Schlammrückführung 2 - Ansteuerung Auf
      A_ZEN_Res_16_1 : Bool;   // Reserve
      A_ZEN_Res_16_2 : Bool;   // Reserve
      A_ZEN_Res_16_3 : Bool;   // Reserve
      A_ZEN_Res_16_4 : Bool;   // Reserve
      A_ZEN_Res_16_5 : Bool;   // Reserve
      A_ZEN_Res_16_6 : Bool;   // Reserve
      A_ZEN_Res_16_7 : Bool;   // Reserve
      A_Zulauf_AS_Auf : Bool;   // Zulauf - Vorlagebehälter - Absperrschieber - Ansteuerung Auf
      A_Zulauf_AS_Zu : Bool;   // Zulauf - Vorlagebehälter - Absperrschieber - Ansteuerung Zu
      A_ZEN_Res_17_2 : Bool;   // Reserve
      A_ZEN_Res_17_3 : Bool;   // Reserve
      A_ZEN_Res_17_4 : Bool;   // Reserve
      A_ZEN_Res_17_5 : Bool;   // Reserve
      A_ZEN_Res_17_6 : Bool;   // Reserve
      A_ZEN_Res_17_7 : Bool;   // Reserve
      E_Zulauf_RA_SA_Ein : Bool;   // Zulauf - Rechen - Sieb - Betrieb
      E_Zulauf_RA_HZS_Ein : Bool;   // Zulauf - Rechen - HZS - Betrieb
      E_Zulauf_RA_VKS_Ein : Bool;   // Zulauf - Rechen - VKS - Betrieb
      E_Zulauf_RA_V_Ein : Bool;   // Zulauf - Rechen - Belüfter - Betrieb
      E_Zulauf_RA_RP_Ein : Bool;   // Zulauf - Rechen - Räumpaddel - Betrieb
      E_Zulauf_RA_FP_Ein : Bool;   // Zulauf - Rechen - Fettpumpe - Betrieb
      E_Zulauf_RA_SA_St : Bool;   // Zulauf - Rechen - Sieb - Störung
      E_Zulauf_RA_HZS_St : Bool;   // Zulauf - Rechen - HZS - Störung
      E_Zulauf_RA_VKS_St : Bool;   // Zulauf - Rechen - VKS - Störung
      E_Zulauf_RA_V_St : Bool;   // Zulauf - Rechen - Belüfter - Störung
      E_Zulauf_RA_RP_St : Bool;   // Zulauf - Rechen - Räumpaddel - Störung
      E_Zulauf_RA_FP_St : Bool;   // Zulauf - Rechen - Fettpumpe - Störung
      E_Zulauf_RA_24V_St : Bool;   // Zulauf - Rechen - Versorgungsspannung 24V - Störung
      E_Zulauf_RA_US_St : Bool;   // Zulauf - Rechen - Ultraschallmessung - Störung
      E_Zulauf_RA_230V_St : Bool;   // Zulauf - Rechen - Versorgungsspannung 230V - Störung
      E_Zulauf_DF_ZI : Bool;   // Zulauf - Rechen - Durchfluss - Impuls
      E_Zulauf_DF_St : Bool;   // Zulauf - Rechen - Durchfluss - Störung
      E_Zulauf_Niv_St : Bool;   // Zulauf - Vorlagebehälter - Niveau - Störung
      E_Verteiler_pH_St : Bool;   // Zulauf - Verteiler - pH-Wert - Störung
      E_Zulauf_AS_EA : Bool;   // Zulauf - Vorlagebehälter - Absperrschieber - Endlage Auf
      E_Zulauf_AS_EZ : Bool;   // Zulauf - Vorlagebehälter - Absperrschieber - Endlage Zu
      E_Zulauf_AS_St : Bool;   // Zulauf - Vorlagebehälter - Absperrschieber - Störung
      E_Zulauf_AS_Bed_vOrt : Bool;   // Zulauf - Vorlagebehälter - Absperrschieber - vor-Ort-Hand
      E_Zulauf_AS_Bed_Fern : Bool;   // Zulauf - Vorlagebehälter - Absperrschieber - vor-Ort-Fern
      E_Zulauf_AS_AF_St : Bool;   // Zulauf - Vorlagebehälter - Absperrschieber - Steuersicherung ausgelöst
      E_ZEN_Res_31_1 : Bool;   // Reserve
      E_ZEN_Res_31_2 : Bool;   // Reserve
      E_ZEN_Res_31_3 : Bool;   // Reserve
      E_ZEN_Res_31_4 : Bool;   // Reserve
      E_ZEN_Res_31_5 : Bool;   // Reserve
      E_ZEN_Res_31_6 : Bool;   // Reserve
      E_ZEN_Res_31_7 : Bool;   // Reserve
      E_ZEN_Res_40_0 : Bool;   // Reserve
      E_Schlamm_BP_Ein : Bool;   // Schlamm - Beschickungspumpe Schlammbeete - Betrieb
      E_Schlamm_BP_St : Bool;   // Schlamm - Beschickungspumpe Schlammbeete - Störung
      E_Schlamm_BP_Bed_vOrt : Bool;   // Schlamm - Beschickungspumpe Schlammbeete - vor-Ort-Hand
      E_Schlamm_BP_Bed_Fern : Bool;   // Schlamm - Beschickungspumpe Schlammbeete - vor-Ort-Fern
      E_Schlamm_BP_AF_St : Bool;   // Schlamm - Beschickungspumpe Schlammbeete - Steuersicherung ausgelöst
      E_Truebwasser_P1_Ein : Bool;   // Trübwasserpumpwerk - Pumpe 1 - Betrieb
      E_Truebwasser_P1_St : Bool;   // Trübwasserpumpwerk - Pumpe 1 - Störung
      E_Truebwasser_P1_Bed_vOrt : Bool;   // Trübwasserpumpwerk - Pumpe 1 - vor-Ort-Hand
      E_Truebwasser_P1_Bed_Fern : Bool;   // Trübwasserpumpwerk - Pumpe 1 - vor-Ort-Fern
      E_Truebwasser_P1_AF_St : Bool;   // Trübwasserpumpwerk - Pumpe 1 - Steuersicherung ausgelöst
      E_Truebwasser_P2_Ein : Bool;   // Trübwasserpumpwerk - Pumpe 2 - Betrieb
      E_Truebwasser_P2_St : Bool;   // Trübwasserpumpwerk - Pumpe 2 - Störung
      E_Truebwasser_P2_Bed_vOrt : Bool;   // Trübwasserpumpwerk - Pumpe 2 - vor-Ort-Hand
      E_Truebwasser_P2_Bed_Fern : Bool;   // Trübwasserpumpwerk - Pumpe 2 - vor-Ort-Fern
      E_Truebwasser_P2_AF_St : Bool;   // Trübwasserpumpwerk - Pumpe 2 - Steuersicherung ausgelöst
      E_Schlamm_AS_EA : Bool;   // Schlamm - Absperrschieber Schlammbeete - Endlage Auf
      E_Schlamm_AS_EZ : Bool;   // Schlamm - Absperrschieber Schlammbeete - Endlage Zu
      E_Schlamm_AS_St : Bool;   // Schlamm - Absperrschieber Schlammbeete - Störung
      E_Schlamm_AS_Bed_vOrt : Bool;   // Schlamm - Absperrschieber Schlammbeete - vor-Ort-Hand
      E_Schlamm_AS_Bed_Fern : Bool;   // Schlamm - Absperrschieber Schlammbeete - vor-Ort-Fern
      E_Schlamm_AS_AF_St : Bool;   // Schlamm - Absperrschieber Schlammbeete - Steuersicherung ausgelöst
      E_ZEN_Res_42_6 : Bool;   // Reserve
      E_ZEN_Res_42_7 : Bool;   // Reserve
      E_Schlamm_Besch_DF_ZI : Bool;   // Schlamm - Beschickung - Durchfluss - Impuls
      E_Schlamm_Besch_DF_St : Bool;   // Schlamm - Beschickung - Durchfluss - Störung
      E_Truebwasser_Niv_St : Bool;   // Trübwasserpumpwerk - Niveau - Störung
      E_Truebwasser_DF_ZI : Bool;   // Trübwasserpumpwerk - Durchfluss - Impuls
      E_Truebwasser_DF_St : Bool;   // Trübwasserpumpwerk - Durchfluss - Störung
      E_ZEN_Res_43_5 : Bool;   // Reserve
      E_ZEN_Res_43_6 : Bool;   // Reserve
      E_ZEN_Res_43_7 : Bool;   // Reserve
      A_Schlamm_BP_Ein : Bool;   // Schlamm - Beschickungspumpe Schlammbeete - Ansteuerung Ein
      A_Truebwasser_P1_Ein : Bool;   // Trübwasserpumpwerk - Pumpe 1 - Ansteuerung Ein
      A_Truebwasser_P2_Ein : Bool;   // Trübwasserpumpwerk - Pumpe 2 - Ansteuerung Ein
      A_Schlamm_AS_Auf : Bool;   // Schlamm - Absperrschieber Schlammbeete - Ansteuerung Auf
      A_Schlamm_AS_Zu : Bool;   // Schlamm - Absperrschieber Schlammbeete - Ansteuerung Zu
      A_ZEN_Res_40_5 : Bool;   // Reserve
      A_ZEN_Res_40_6 : Bool;   // Reserve
      A_ZEN_Res_40_7 : Bool;   // Reserve
      A_ZEN_Res_41_0 : Bool;   // Reserve
      A_ZEN_Res_41_1 : Bool;   // Reserve
      A_ZEN_Res_41_2 : Bool;   // Reserve
      A_ZEN_Res_41_3 : Bool;   // Reserve
      A_ZEN_Res_41_4 : Bool;   // Reserve
      A_ZEN_Res_41_5 : Bool;   // Reserve
      A_ZEN_Res_41_6 : Bool;   // Reserve
      A_ZEN_Res_41_7 : Bool;   // Reserve
      A_ZEN_Res_42_0 : Bool;   // Reserve
      A_ZEN_Res_42_1 : Bool;   // Reserve
      A_ZEN_Res_42_2 : Bool;   // Reserve
      A_ZEN_Res_42_3 : Bool;   // Reserve
      A_ZEN_Res_42_4 : Bool;   // Reserve
      A_ZEN_Res_42_5 : Bool;   // Reserve
      A_ZEN_Res_42_6 : Bool;   // Reserve
      A_ZEN_Res_42_7 : Bool;   // Reserve
      A_ZEN_Res_43_0 : Bool;   // Reserve
      A_ZEN_Res_43_1 : Bool;   // Reserve
      A_ZEN_Res_43_2 : Bool;   // Reserve
      A_ZEN_Res_43_3 : Bool;   // Reserve
      A_ZEN_Res_43_4 : Bool;   // Reserve
      A_ZEN_Res_43_5 : Bool;   // Reserve
      A_ZEN_Res_43_6 : Bool;   // Reserve
      A_ZEN_Res_43_7 : Bool;   // Reserve
      ZEN_DiagKom_IEC : Bool;   // Diagnose Kommunikation - Störung Kopplung zu Fernwirkzentrale
      ZEN_DiagKom_DP_BF3 : Bool;   // Diagnose Kommunikation - Busfehler Teilnehmer 3 - UV Gebläsestation
      ZEN_DiagKom_DP_BF4 : Bool;   // Diagnose Kommunikation - Busfehler Teilnehmer 4 - UV Alte Hebestelle
      ZEN_DiagKom_DP_BF5 : Bool;   // Diagnose Kommunikation - Busfehler Teilnehmer 5 - Reserve
      ZEN_DiagKom_DP_BF6 : Bool;   // Diagnose Kommunikation - Busfehler Teilnehmer 6 - Reserve
      ZEN_DiagKom_DP_BF7 : Bool;   // Diagnose Kommunikation - Busfehler Teilnehmer 7 - Reserve
      ZEN_DiagKom_DP_BF8 : Bool;   // Diagnose Kommunikation - Busfehler Teilnehmer 8 - Reserve
      ZEN_DiagKom_DP_BF9 : Bool;   // Diagnose Kommunikation - Busfehler Teilnehmer 9 - Reserve
      ZEN_DiagKom_DP_BF10 : Bool;   // Diagnose Kommunikation - Busfehler Teilnehmer 10 - Reserve
      ZEN_DiagKom_DP_BF11 : Bool;   // Diagnose Kommunikation - Busfehler Teilnehmer 11 - Reserve
      ZEN_DiagKom_DP_BF12 : Bool;   // Diagnose Kommunikation - Busfehler Teilnehmer 12 - Reserve
      ZEN_DiagKom_DP_BF13 : Bool;   // Diagnose Kommunikation - Busfehler Teilnehmer 13 - Reserve
      ZEN_DiagKom_DP_BF14 : Bool;   // Diagnose Kommunikation - Busfehler Teilnehmer 14 - Reserve
      ZEN_DiagKom_DP_BF15 : Bool;   // Diagnose Kommunikation - Busfehler Teilnehmer 15 - Reserve
      ZEN_DiagKom_DP_BF16 : Bool;   // Diagnose Kommunikation - Busfehler Teilnehmer 16 - Reserve
      ZEN_DiagKom_DP_BF17 : Bool;   // Diagnose Kommunikation - Busfehler Teilnehmer 17 - Reserve
      ZEN_ObjS_Begehung : Bool;   // Betriebsgebäude - Objektschutz - Begehung
      ZEN_ObjS_Alarm : Bool;   // Betriebsgebäude - Objektschutz - Alarm
      ZEN_ObjS_unscharf : Bool;   // Betriebsgebäude - Objektschutz - unscharf
      ZEN_ObjS_scharf : Bool;   // Betriebsgebäude - Objektschutz - Scharfschaltung
      ZEN_NA_res : Bool;   // UV BG - Netzausfall
      ZEN_Bed_aktiv : Bool;   // UV BG Bedienstelle - Bediener aktiv
      ZEN_Res_DB100_40_6 : Bool;   // Reserve
      ZEN_Res_DB100_40_7 : Bool;   // Reserve
      BB_Auto_GeblW_G1_B1 : Bool;   // Steuerung Belüftung - Automatik - Vorwahl Gebläse 1 auf Becken 1
      BB_Auto_GeblW_G2_B2 : Bool;   // Steuerung Belüftung - Automatik - Vorwahl Gebläse 2 auf Becken 2
      BB_Auto_GeblW_G3_B1 : Bool;   // Steuerung Belüftung - Automatik - Vorwahl Gebläse 3 auf Becken 1
      BB_Auto_GeblW_G3_B2 : Bool;   // Steuerung Belüftung - Automatik - Vorwahl Gebläse 3 auf Becken 2
      ZEN_Res_DB100_41_4 : Bool;   // Reserve
      ZEN_Res_DB100_41_5 : Bool;   // Reserve
      ZEN_Res_DB100_41_6 : Bool;   // Reserve
      ZEN_Res_DB100_41_7 : Bool;   // Reserve
      Biocos1_BA_SU_RB : Bool;   // Steuerung Biocos 1 - Betriebsart - Schaltuhrbetrieb - Rückmeldung
      Biocos1_BA_P1_RB : Bool;   // Steuerung Biocos 1 - Betriebsart - Parametersatz 1 - Rückmeldung
      Biocos1_BA_P2_RB : Bool;   // Steuerung Biocos 1 - Betriebsart - Parametersatz 2 - Rückmeldung
      Biocos1_BA_Aus_RB : Bool;   // Steuerung Biocos 1 - Betriebsart - Aus - Rückmeldung
      Biocos1_Auto_P1_aktiv : Bool;   // Steuerung Biocos 1 - Automatik - Parametersatz 1 aktiv
      Biocos1_Auto_P2_aktiv : Bool;   // Steuerung Biocos 1 - Automatik - Parametersatz 2 aktiv
      Biocos1_Auto_Bel_O2_Ein_RB : Bool;   // Steuerung Biocos 1 - Automatik - Belüftung nach O2-Gehalt aktiv
      Biocos1_Auto_Bel_O2_Aus_RB : Bool;   // Steuerung Biocos 1 - Automatik - Belüftung nach O2-Gehalt aus -> Intervallbelüftung
      Biocos1_Auto_Bel_O2_St : Bool;   // Steuerung Biocos 1 - Automatik - Störung Messung O2-Gehalt -> Intervallbelüftung
      Biocos1_Auto_Bel_O2_min : Bool;   // Steuerung Biocos 1 - Automatik - Belüftung nach O2-Gehalt -> min.-Wert nicht erreicht
      Biocos1_Auto_UeSS_Menge_Ein_RB : Bool;   // Steuerung Biocos 1 - Automatik - ÜSS-Abzug nach Menge aktiv
      Biocos1_Auto_UeSS_Menge_Aus_RB : Bool;   // Steuerung Biocos 1 - Automatik - ÜSS-Abzug nach Menge aus -> Zeit
      Biocos1_Auto_UeSS_Menge_St : Bool;   // Steuerung Biocos 1 - Automatik - ÜSS-Abzug nach Menge -> Zeitüberschreitung
      ZEN_Res_DB100_43_5 : Bool;   // Reserve
      ZEN_Res_DB100_43_6 : Bool;   // Reserve
      ZEN_Res_DB100_43_7 : Bool;   // Reserve
      Biocos1_Auto_Bel_Phase : Bool;   // Steuerung Biocos 1 - Automatik - Belüftungsphase aktiv
      Biocos1_Auto_Bel_Verz : Bool;   // Steuerung Biocos 1 - Automatik - Verzögerung bis Freigabe Belüftung
      Biocos1_Auto_Bel_Frg : Bool;   // Steuerung Biocos 1 - Automatik - Freigabe Belüftung
      Biocos1_Auto_Bel_Int : Bool;   // Steuerung Biocos 1 - Automatik - Belüftung im Intervall aktiv
      Biocos1_Auto_UeSS : Bool;   // Steuerung Biocos 1 - Automatik - ÜSS-Abzug aktiv
      ZEN_Res_DB100_44_5 : Bool;   // Reserve
      ZEN_Res_DB100_44_6 : Bool;   // Reserve
      ZEN_Res_DB100_44_7 : Bool;   // Reserve
      Biocos1_Auto_U1 : Bool;   // Steuerung Biocos 1 - Automatik - U-Phase SU-Becken 1 aktiv
      Biocos1_Auto_V1 : Bool;   // Steuerung Biocos 1 - Automatik - V-Phase SU-Becken 1 aktiv
      Biocos1_Auto_A1 : Bool;   // Steuerung Biocos 1 - Automatik - A-Phase SU-Becken 1 aktiv
      Biocos1_Auto_U2 : Bool;   // Steuerung Biocos 1 - Automatik - U-Phase SU-Becken 2 aktiv
      Biocos1_Auto_V2 : Bool;   // Steuerung Biocos 1 - Automatik - V-Phase SU-Becken 2 aktiv
      Biocos1_Auto_A2 : Bool;   // Steuerung Biocos 1 - Automatik - A-Phase SU-Becken 2 aktiv
      Biocos1_Auto_SR1 : Bool;   // Steuerung Biocos 1 - Automatik - Schlammrückführung SU-Becken 1 aktiv
      Biocos1_Auto_SR2 : Bool;   // Steuerung Biocos 1 - Automatik - Schlammrückführung SU-Becken 2 aktiv
      Biocos2_BA_SU_RB : Bool;   // Steuerung Biocos 2 - Betriebsart - Schaltuhrbetrieb - Rückmeldung
      Biocos2_BA_P1_RB : Bool;   // Steuerung Biocos 2 - Betriebsart - Parametersatz 1 - Rückmeldung
      Biocos2_BA_P2_RB : Bool;   // Steuerung Biocos 2 - Betriebsart - Parametersatz 2 - Rückmeldung
      Biocos2_BA_Aus_RB : Bool;   // Steuerung Biocos 2 - Betriebsart - Aus - Rückmeldung
      Biocos2_Auto_P1_aktiv : Bool;   // Steuerung Biocos 2 - Automatik - Parametersatz 1 aktiv
      Biocos2_Auto_P2_aktiv : Bool;   // Steuerung Biocos 2 - Automatik - Parametersatz 2 aktiv
      Biocos2_Auto_Bel_O2_Ein_RB : Bool;   // Steuerung Biocos 2 - Automatik - Belüftung nach O2-Gehalt aktiv
      Biocos2_Auto_Bel_O2_Aus_RB : Bool;   // Steuerung Biocos 2 - Automatik - Belüftung nach O2-Gehalt aus -> Intervallbelüftung
      Biocos2_Auto_Bel_O2_St : Bool;   // Steuerung Biocos 2 - Automatik - Störung Messung O2-Gehalt -> Intervallbelüftung
      Biocos2_Auto_Bel_O2_min : Bool;   // Steuerung Biocos 2 - Automatik - Belüftung nach O2-Gehalt -> min.-Wert nicht erreicht
      Biocos2_Auto_UeSS_Menge_Ein_RB : Bool;   // Steuerung Biocos 2 - Automatik - ÜSS-Abzug nach Menge aktiv
      Biocos2_Auto_UeSS_Menge_Aus_RB : Bool;   // Steuerung Biocos 2 - Automatik - ÜSS-Abzug nach Menge aus -> Zeit
      Biocos2_Auto_UeSS_Menge_St : Bool;   // Steuerung Biocos 2 - Automatik - ÜSS-Abzug nach Menge -> Zeitüberschreitung
      ZEN_Res_DB100_47_5 : Bool;   // Reserve
      ZEN_Res_DB100_47_6 : Bool;   // Reserve
      ZEN_Res_DB100_47_7 : Bool;   // Reserve
      Biocos2_Auto_Bel_Phase : Bool;   // Steuerung Biocos 2 - Automatik - Belüftungsphase aktiv
      Biocos2_Auto_Bel_Verz : Bool;   // Steuerung Biocos 2 - Automatik - Verzögerung bis Freigabe Belüftung
      Biocos2_Auto_Bel_Frg : Bool;   // Steuerung Biocos 2 - Automatik - Freigabe Belüftung
      Biocos2_Auto_Bel_Int : Bool;   // Steuerung Biocos 2 - Automatik - Belüftung im Intervall aktiv
      Biocos2_Auto_UeSS : Bool;   // Steuerung Biocos 2 - Automatik - ÜSS-Abzug aktiv
      ZEN_Res_DB100_48_5 : Bool;   // Reserve
      ZEN_Res_DB100_48_6 : Bool;   // Reserve
      ZEN_Res_DB100_48_7 : Bool;   // Reserve
      Biocos2_Auto_U1 : Bool;   // Steuerung Biocos 2 - Automatik - U-Phase SU-Becken 1 aktiv
      Biocos2_Auto_V1 : Bool;   // Steuerung Biocos 2 - Automatik - V-Phase SU-Becken 1 aktiv
      Biocos2_Auto_A1 : Bool;   // Steuerung Biocos 2 - Automatik - A-Phase SU-Becken 1 aktiv
      Biocos2_Auto_U2 : Bool;   // Steuerung Biocos 2 - Automatik - U-Phase SU-Becken 2 aktiv
      Biocos2_Auto_V2 : Bool;   // Steuerung Biocos 2 - Automatik - V-Phase SU-Becken 2 aktiv
      Biocos2_Auto_A2 : Bool;   // Steuerung Biocos 2 - Automatik - A-Phase SU-Becken 2 aktiv
      Biocos2_Auto_SR1 : Bool;   // Steuerung Biocos 2 - Automatik - Schlammrückführung SU-Becken 1 aktiv
      Biocos2_Auto_SR2 : Bool;   // Steuerung Biocos 2 - Automatik - Schlammrückführung SU-Becken 2 aktiv
      ZEN_Res_DB100_50_0 : Bool;   // Reserve
      ZEN_Res_DB100_50_1 : Bool;   // Reserve
      ZEN_Res_DB100_50_2 : Bool;   // Reserve
      ZEN_Res_DB100_50_3 : Bool;   // Reserve
      ZEN_Res_DB100_50_4 : Bool;   // Reserve
      ZEN_Res_DB100_50_5 : Bool;   // Reserve
      ZEN_Res_DB100_50_6 : Bool;   // Reserve
      ZEN_Res_DB100_50_7 : Bool;   // Reserve
      ZEN_Res_DB100_51_0 : Bool;   // Reserve
      ZEN_Res_DB100_51_1 : Bool;   // Reserve
      ZEN_Res_DB100_51_2 : Bool;   // Reserve
      ZEN_Res_DB100_51_3 : Bool;   // Reserve
      ZEN_Res_DB100_51_4 : Bool;   // Reserve
      ZEN_Res_DB100_51_5 : Bool;   // Reserve
      ZEN_Res_DB100_51_6 : Bool;   // Reserve
      ZEN_Res_DB100_51_7 : Bool;   // Reserve
      IEC_Meld_LS_001 : Bool;   // Sammelmeldung an Leitstelle - Gebläse 1 Störung
      IEC_Meld_LS_002 : Bool;   // Sammelmeldung an Leitstelle - Gebläse 2 Störung
      IEC_Meld_LS_003 : Bool;   // Sammelmeldung an Leitstelle - Gebläse 3 Störung
      IEC_Meld_LS_004 : Bool;   // Sammelmeldung an Leitstelle - Belebungsbecken 1 Rezipumpe 1 Störung
      IEC_Meld_LS_005 : Bool;   // Sammelmeldung an Leitstelle - Belebungsbecken 1 Rezipumpe 2 Störung
      IEC_Meld_LS_006 : Bool;   // Sammelmeldung an Leitstelle - Belebungsbecken 1 Überschussschlammpumpe Störung
      IEC_Meld_LS_007 : Bool;   // Sammelmeldung an Leitstelle - Belebungsbecken 1 Ablaufschieber Störung
      IEC_Meld_LS_008 : Bool;   // Sammelmeldung an Leitstelle - Belebungsbecken 1 Schlammrückführung Störung
      IEC_Meld_LS_009 : Bool;   // Sammelmeldung an Leitstelle - Belebungsbecken 2 Rezipumpe 1 Störung
      IEC_Meld_LS_010 : Bool;   // Sammelmeldung an Leitstelle - Belebungsbecken 2 Rezipumpe 2 Störung
      IEC_Meld_LS_011 : Bool;   // Sammelmeldung an Leitstelle - Belebungsbecken 2 Überschussschlammpumpe Störung
      IEC_Meld_LS_012 : Bool;   // Sammelmeldung an Leitstelle - Belebungsbecken 2 Ablaufschieber Störung
      IEC_Meld_LS_013 : Bool;   // Sammelmeldung an Leitstelle - Belebungsbecken 2 Schlammrückführung Störung
      IEC_Meld_LS_014 : Bool;   // Sammelmeldung an Leitstelle - Rechenanlage Störung
      IEC_Meld_LS_015 : Bool;   // Sammelmeldung an Leitstelle - Schlammpumpe Störung
      IEC_Meld_LS_016 : Bool;   // Sammelmeldung an Leitstelle - Eindicker Störung
      IEC_Meld_LS_017 : Bool;   // Sammelmeldung an Leitstelle - Trübwasserpumpe Störung
      IEC_Meld_LS_018 : Bool;   // Sammelmeldung an Leitstelle - Schlammstapelbehälter Störung
      IEC_Meld_LS_019 : Bool;   // Sammelmeldung an Leitstelle - Druckluftkompressor Störung
      IEC_Meld_LS_020 : Bool;   // Sammelmeldung an Leitstelle - Zulaufschieber Störung
      IEC_Meld_LS_021 : Bool;   // Sammelmeldung an Leitstelle - Luftschieber Störung
      IEC_Meld_LS_022 : Bool;   // Sammelmeldung an Leitstelle - Filtration Störung
      IEC_Meld_LS_023 : Bool;   // Sammelmeldung an Leitstelle - Reserve 23
      IEC_Meld_LS_024 : Bool;   // Sammelmeldung an Leitstelle - Netzausfall
      IEC_Meld_LS_025 : Bool;   // Sammelmeldung an Leitstelle - 400VAC/24VDC Sammelstörung
      IEC_Meld_LS_026 : Bool;   // Sammelmeldung an Leitstelle - Mengenmessung Störung
      IEC_Meld_LS_027 : Bool;   // Sammelmeldung an Leitstelle - Biologie Sammelstörung
      IEC_Meld_LS_028 : Bool;   // Sammelmeldung an Leitstelle - Belebungsbecken 1 Biologie Störung
      IEC_Meld_LS_029 : Bool;   // Sammelmeldung an Leitstelle - Belebungsbecken 2 Biologie Störung
      IEC_Meld_LS_030 : Bool;   // Sammelmeldung an Leitstelle - Höhenstände Pumpwerke Störung
      IEC_Meld_LS_031 : Bool;   // Sammelmeldung an Leitstelle - Höhenstände Kläranlage Störung
      IEC_Meld_LS_032 : Bool;   // Sammelmeldung an Leitstelle - Türkontakt/Alarmanlage
      Zulauf_PW_BA_Auto_RB : Bool;   // Steuerung Zulauf/Freigabe Pumpwerke - Betriebsart - Automatik - Rückmeldung
      Zulauf_PW_BA_Aus_RB : Bool;   // Steuerung Zulauf/Freigabe Pumpwerke - Betriebsart - Aus - Rückmeldung
      Zulauf_PW_Auto_DF_max : Bool;   // Steuerung Zulauf/Freigabe Pumpwerke - Automatik - Grenzwert max. Durchflußmenge durch die KA
      Zulauf_PW_Auto_Niv_max : Bool;   // Steuerung Zulauf/Freigabe Pumpwerke - Automatik - Niveau Vorlageschacht Zulauf - alle Freigaben ext. PW abschalten
      Zulauf_PW_Auto_Niv_AS : Bool;   // Steuerung Zulauf/Freigabe Pumpwerke - Automatik - Niveau Vorlageschacht Zulauf - Freigabe ext. PW zyklisch abschalten
      Zulauf_PW_Auto_Niv_ZS : Bool;   // Steuerung Zulauf/Freigabe Pumpwerke - Automatik - Niveau Vorlageschacht Zulauf - Freigabe ext. PW zyklisch zuschalten
      Zulauf_PW_Auto_Niv_min : Bool;   // Steuerung Zulauf/Freigabe Pumpwerke - Automatik - Niveau Vorlageschacht Zulauf - alle Freigaben ext. PW zuschalten
      Zulauf_PW_Auto_Frg_Ein : Bool;   // Steuerung Zulauf/Freigabe Pumpwerke - Status - alle Freigaben eingeschaltet
      Zulauf_PW_Auto_Frg_TeilAus : Bool;   // Steuerung Zulauf/Freigabe Pumpwerke - Status - mindestens eine Freigabe abgeschaltet
      Zulauf_PW_Auto_Frg_Aus : Bool;   // Steuerung Zulauf/Freigabe Pumpwerke - Status - alle Freigaben ausgeschaltet
      ZEN_Res_DB100_57_2 : Bool;   // Reserve
      Zulauf_RA_SA_Stillst : Bool;   // Zulauf - Rechen - Sieb - Stillstand länger als 2h
      ZEN_Res_DB100_57_4 : Bool;   // Reserve
      ZEN_Res_DB100_57_5 : Bool;   // Reserve
      ZEN_Res_DB100_57_6 : Bool;   // Reserve
      ZEN_Res_DB100_57_7 : Bool;   // Reserve
      Schlamm_TW_BA_Auto_RB : Bool;   // Steuerung Trübwasserpumpwerk - Betriebsart - Automatik - Rückmeldung
      Schlamm_TW_BA_Aus_RB : Bool;   // Steuerung Trübwasserpumpwerk - Betriebsart - Aus - Rückmeldung
      Schlamm_TW_Auto_Frg_Zt : Bool;   // Steuerung Trübwasserpumpwerk - Automatik - Freigabe Abzug (Uhrzeit)
      Schlamm_TW_Auto_2P_Ein : Bool;   // Steuerung Trübwasserpumpwerk - Automatik - Niveau Trübwasserschacht - Abpumpen 2 Pumpen Ein
      Schlamm_TW_Auto_1P_Ein : Bool;   // Steuerung Trübwasserpumpwerk - Automatik - Niveau Trübwasserschacht - Abpumpen 1 Pumpe Ein
      ZEN_Res_DB100_58_5 : Bool;   // Reserve
      ZEN_Res_DB100_58_6 : Bool;   // Reserve
      ZEN_Res_DB100_58_7 : Bool;   // Reserve
      Schlamm_Besch_BA_Auto_RB : Bool;   // Steuerung Beschickung Schlammbeete - Betriebsart - Automatik - Rückmeldung
      Schlamm_Besch_BA_Aus_RB : Bool;   // Steuerung Beschickung Schlammbeete - Betriebsart - Aus - Rückmeldung
      Schlamm_Besch_Auto_Zt_max : Bool;   // Steuerung Beschickung Schlammbeete - Automatik - Überwachung Zeitüberschreitung
      ZEN_Res_DB100_59_3 : Bool;   // Reserve
      ZEN_Res_DB100_59_4 : Bool;   // Reserve
      ZEN_Res_DB100_59_5 : Bool;   // Reserve
      ZEN_Res_DB100_59_6 : Bool;   // Reserve
      ZEN_Res_DB100_59_7 : Bool;   // Reserve
      PO4_Elim_BA_Auto_RB : Bool;   // Steuerung PO4-Elimination - Betriebsart - Automatik - Rückmeldung
      PO4_Elim_BA_Hand_RB : Bool;   // Steuerung PO4-Elimination - Betriebsart - Handvorgabe - Rückmeldung
      PO4_Elim_BA_Aus_RB : Bool;   // Steuerung PO4-Elimination - Betriebsart - Aus - Rückmeldung
      PO4_Elim_Auto_P_Ein : Bool;   // Steuerung PO4-Elimination - Automatik - Anforderung Dosierpumpe
      PO4_Elim_SC_Status_W1 : Bool;   // Steuerung PO4-Elimination - Status Dosierrechner Hach-Lange - Sammelmeldung Warnung I
      PO4_Elim_SC_Status_W2 : Bool;   // Steuerung PO4-Elimination - Status Dosierrechner Hach-Lange - Sammelmeldung Warnung II
      PO4_Elim_SC_Status_DevE : Bool;   // Steuerung PO4-Elimination - Status Dosierrechner Hach-Lange - Sammelmeldung Device Error
      PO4_Elim_SC_Status_CE : Bool;   // Steuerung PO4-Elimination - Status Dosierrechner Hach-Lange - Sammelmeldung Classified Error
      Biocos1_BA_O2_Reg_FW_RB : Bool;   // Steuerung Biocos 1 - Betriebsart O2-Regler - Festwert - Rückmeldung
      Biocos1_BA_O2_Reg_Auto_RB : Bool;   // Steuerung Biocos 1 - Betriebsart O2-Regler - Automatik - Rückmeldung
      Biocos1_Auto_Bel_O2_Reg_St : Bool;   // Steuerung Biocos 1 - Automatik O2-Regler - Störung Messung O2-Gehalt -> Belüftung nach Festwert
      Biocos1_Auto_Bel_O2_Reg_GW_max : Bool;   // Steuerung Biocos 1 - Automatik O2-Regler - Sollwert O2-Gehalt max -> Abschaltung Gebläse
      ZEN_Res_DB100_61_4 : Bool;   // Reserve
      ZEN_Res_DB100_61_5 : Bool;   // Reserve
      ZEN_Res_DB100_61_6 : Bool;   // Reserve
      ZEN_Res_DB100_61_7 : Bool;   // Reserve
      Biocos2_BA_O2_Reg_FW_RB : Bool;   // Steuerung Biocos 2 - Betriebsart O2-Regler - Festwert - Rückmeldung
      Biocos2_BA_O2_Reg_Auto_RB : Bool;   // Steuerung Biocos 2 - Betriebsart O2-Regler - Automatik - Rückmeldung
      Biocos2_Auto_Bel_O2_Reg_St : Bool;   // Steuerung Biocos 2 - Automatik O2-Regler - Störung Messung O2-Gehalt -> Belüftung nach Festwert
      Biocos2_Auto_Bel_O2_Reg_GW_max : Bool;   // Steuerung Biocos 2 - Automatik O2-Regler - Sollwert O2-Gehalt max -> Abschaltung Gebläse
      ZEN_Res_DB100_62_4 : Bool;   // Reserve
      ZEN_Res_DB100_62_5 : Bool;   // Reserve
      ZEN_Res_DB100_62_6 : Bool;   // Reserve
      ZEN_Res_DB100_62_7 : Bool;   // Reserve
      ZEN_Res_DB100_63_0 : Bool;   // Reserve
      ZEN_Res_DB100_63_1 : Bool;   // Reserve
      ZEN_Res_DB100_63_2 : Bool;   // Reserve
      ZEN_Res_DB100_63_3 : Bool;   // Reserve
      ZEN_Res_DB100_63_4 : Bool;   // Reserve
      ZEN_Res_DB100_63_5 : Bool;   // Reserve
      ZEN_Res_DB100_63_6 : Bool;   // Reserve
      ZEN_Res_DB100_63_7 : Bool;   // Reserve
      BB_G1_KS_AM9 : Bool;   // Belebung - SigmaControl Gebläse 1 - Alarme - Zulässige Innentemperatur von SIGMA CONTROL 2 MCS oder IOM überschritten
      BB_G1_KS_AM10 : Bool;   // Belebung - SigmaControl Gebläse 1 - Alarme - Enddruck p2 zu hoch
      BB_G1_KS_AM11 : Bool;   // Belebung - SigmaControl Gebläse 1 - Alarme - Reserve
      BB_G1_KS_AM12 : Bool;   // Belebung - SigmaControl Gebläse 1 - Alarme - Reserve
      BB_G1_KS_AM13 : Bool;   // Belebung - SigmaControl Gebläse 1 - Alarme - Überlast Gebläsemotor -> Abschaltung wegen Überlastung
      BB_G1_KS_AM14 : Bool;   // Belebung - SigmaControl Gebläse 1 - Alarme - Abschaltung des Nachkühler-Lüfters wegen Überlastung
      BB_G1_KS_AM15 : Bool;   // Belebung - SigmaControl Gebläse 1 - Alarme - Maximal zulässige Verdichtungs-Endtemperatur (VET) überschritten
      BB_G1_KS_AM16 : Bool;   // Belebung - SigmaControl Gebläse 1 - Alarme - Reserve
      BB_G1_KS_AM1 : Bool;   // Belebung - SigmaControl Gebläse 1 - Alarme - Reserve
      BB_G1_KS_AM2 : Bool;   // Belebung - SigmaControl Gebläse 1 - Alarme - Temperatur Gebläsemotor zu hoch
      BB_G1_KS_AM3 : Bool;   // Belebung - SigmaControl Gebläse 1 - Alarme - Reserve
      BB_G1_KS_AM4 : Bool;   // Belebung - SigmaControl Gebläse 1 - Alarme - NOT-HALT-Befehlsgerät betätigt
      BB_G1_KS_AM5 : Bool;   // Belebung - SigmaControl Gebläse 1 - Alarme - Schmierölstand Antriebsseite Gebläseblock zu niedrig
      BB_G1_KS_AM6 : Bool;   // Belebung - SigmaControl Gebläse 1 - Alarme - Schmierölstand Steuerseite Gebläseblock zu niedrig
      BB_G1_KS_AM7 : Bool;   // Belebung - SigmaControl Gebläse 1 - Alarme - Phasenfehler oder Unter-/Überspannung Gebläsemotor
      BB_G1_KS_AM8 : Bool;   // Belebung - SigmaControl Gebläse 1 - Alarme - Diagnose-Sammelmeldung
      BB_G1_KS_AM25 : Bool;   // Belebung - SigmaControl Gebläse 1 - Alarme - Sammelfehler IOM
      BB_G1_KS_AM26 : Bool;   // Belebung - SigmaControl Gebläse 1 - Alarme - Reserve
      BB_G1_KS_AM27 : Bool;   // Belebung - SigmaControl Gebläse 1 - Alarme - Filter verstopft -> Verschmutzung des Ansaugfilters
      BB_G1_KS_AM28 : Bool;   // Belebung - SigmaControl Gebläse 1 - Alarme - Öltemperatur t3 sehr hoch
      BB_G1_KS_AM29 : Bool;   // Belebung - SigmaControl Gebläse 1 - Alarme - Reserve
      BB_G1_KS_AM30 : Bool;   // Belebung - SigmaControl Gebläse 1 - Alarme - Reserve
      BB_G1_KS_AM31 : Bool;   // Belebung - SigmaControl Gebläse 1 - Alarme - Temperaturdifferenz t2 (VET) - t1 (Ansaugtemperatur) zu hoch
      BB_G1_KS_AM32 : Bool;   // Belebung - SigmaControl Gebläse 1 - Alarme - Druckverhältnis über Block zu hoch
      BB_G1_KS_AM17 : Bool;   // Belebung - SigmaControl Gebläse 1 - Alarme - Reserve
      BB_G1_KS_AM18 : Bool;   // Belebung - SigmaControl Gebläse 1 - Alarme - Abschaltung des Schalldämmhauben-Lüfters wegen Überlastung
      BB_G1_KS_AM19 : Bool;   // Belebung - SigmaControl Gebläse 1 - Alarme - Ansaugdruck p1 zu niedrig -> Verschmutzung des Ansaugfilters
      BB_G1_KS_AM20 : Bool;   // Belebung - SigmaControl Gebläse 1 - Alarme - Temperatur unter der Schalldämmhaube zu hoch
      BB_G1_KS_AM21 : Bool;   // Belebung - SigmaControl Gebläse 1 - Alarme - Reserve
      BB_G1_KS_AM22 : Bool;   // Belebung - SigmaControl Gebläse 1 - Alarme - Differenzdruck zu hoch
      BB_G1_KS_AM23 : Bool;   // Belebung - SigmaControl Gebläse 1 - Alarme - Ansaugtemperatur t1 zu hoch
      BB_G1_KS_AM24 : Bool;   // Belebung - SigmaControl Gebläse 1 - Alarme - Ansaugtemperatur t1 zu niedrig
      BB_G1_KS_AM41 : Bool;   // Belebung - SigmaControl Gebläse 1 - Alarme - Überspannung im Stromversorgungsnetz
      BB_G1_KS_AM42 : Bool;   // Belebung - SigmaControl Gebläse 1 - Alarme - Fehler am AFxM-Ventil-Aktor
      BB_G1_KS_AM43 : Bool;   // Belebung - SigmaControl Gebläse 1 - Alarme - Reserve
      BB_G1_KS_AM44 : Bool;   // Belebung - SigmaControl Gebläse 1 - Alarme - Blockdrehzahl liegt außerhalb des erlaubten Bereiches -> Fehler im Antriebsmotor oder Keilriemen
      BB_G1_KS_AM45 : Bool;   // Belebung - SigmaControl Gebläse 1 - Alarme - Vibration des Gebläses zu hoch
      BB_G1_KS_AM46 : Bool;   // Belebung - SigmaControl Gebläse 1 - Alarme - Interner Fehler Frequenzumrichter für Gebläsemotor
      BB_G1_KS_AM47 : Bool;   // Belebung - SigmaControl Gebläse 1 - Alarme - Kommunikationsfehler RS485-FC -> USS-Bus Kommunikationsfehler
      BB_G1_KS_AM48 : Bool;   // Belebung - SigmaControl Gebläse 1 - Alarme - Sammelmeldung des Leistungsteils FU
      BB_G1_KS_AM33 : Bool;   // Belebung - SigmaControl Gebläse 1 - Alarme - Reserve
      BB_G1_KS_AM34 : Bool;   // Belebung - SigmaControl Gebläse 1 - Alarme - Reserve
      BB_G1_KS_AM35 : Bool;   // Belebung - SigmaControl Gebläse 1 - Alarme - Druckdifferenz über den Block zu niedrig
      BB_G1_KS_AM36 : Bool;   // Belebung - SigmaControl Gebläse 1 - Alarme - Reserve
      BB_G1_KS_AM37 : Bool;   // Belebung - SigmaControl Gebläse 1 - Alarme - Reserve
      BB_G1_KS_AM38 : Bool;   // Belebung - SigmaControl Gebläse 1 - Alarme - Ansaugdruck p1 zu niedrig -> Verschmutzung des Ansaugfilters
      BB_G1_KS_AM39 : Bool;   // Belebung - SigmaControl Gebläse 1 - Alarme - Enddruck p2 zu hoch
      BB_G1_KS_AM40 : Bool;   // Belebung - SigmaControl Gebläse 1 - Alarme - Netzschütz schaltet nicht aus oder nicht ein
      BB_G1_KS_AM57 : Bool;   // Belebung - SigmaControl Gebläse 1 - Alarme - Schwerlastüberwachung ausgelöst FU -> Schwerlastüberwachung ausgelöst
      BB_G1_KS_AM58 : Bool;   // Belebung - SigmaControl Gebläse 1 - Alarme - p1-Sensor-Fehler Fehler Drucksensor Ansaugseite Gebläseblock
      BB_G1_KS_AM59 : Bool;   // Belebung - SigmaControl Gebläse 1 - Alarme - p2-Sensor-Fehler Fehler Drucksensor Auslassseite Gebläseblock
      BB_G1_KS_AM60 : Bool;   // Belebung - SigmaControl Gebläse 1 - Alarme - Fehler externer Analogeingang Fehler am externen Analogeingang
      BB_G1_KS_AM61 : Bool;   // Belebung - SigmaControl Gebläse 1 - Alarme - t2-Sensor-Fehler Fehler Sensor PT100 Auslasssseite Gebläseblock
      BB_G1_KS_AM62 : Bool;   // Belebung - SigmaControl Gebläse 1 - Alarme - t_S-Sensor-Fehler Fehler Sensor PT100 Schalldämmhaube
      BB_G1_KS_AM63 : Bool;   // Belebung - SigmaControl Gebläse 1 - Alarme - t1-Sensor-Fehler Fehler Sensor PT100 Ansaugseite Gebläseblock
      BB_G1_KS_AM64 : Bool;   // Belebung - SigmaControl Gebläse 1 - Alarme - t_M-Sensor-Fehler Fehler Sensor PT100 Antriebsmotor
      BB_G1_KS_AM49 : Bool;   // Belebung - SigmaControl Gebläse 1 - Alarme - Reserve
      BB_G1_KS_AM50 : Bool;   // Belebung - SigmaControl Gebläse 1 - Alarme - Nachschmiereinrichtung meldet seit längerer Zeit einen Fehler
      BB_G1_KS_AM51 : Bool;   // Belebung - SigmaControl Gebläse 1 - Alarme - Reserve
      BB_G1_KS_AM52 : Bool;   // Belebung - SigmaControl Gebläse 1 - Alarme - Reserve
      BB_G1_KS_AM53 : Bool;   // Belebung - SigmaControl Gebläse 1 - Alarme - Fehler USS Handler FU -> USS Busfehler
      BB_G1_KS_AM54 : Bool;   // Belebung - SigmaControl Gebläse 1 - Alarme - PKW-Anfragen erfolglos FU -> USS Kommunikation gestört
      BB_G1_KS_AM55 : Bool;   // Belebung - SigmaControl Gebläse 1 - Alarme - Fehler FU Einschaltung FU -> Fehler beim Einschalten des Frequenzumrichters
      BB_G1_KS_AM56 : Bool;   // Belebung - SigmaControl Gebläse 1 - Alarme - Motor -> n_min nicht erreicht FU -> Mindestdrehzahl nicht erreicht
      BB_G1_KS_AM73 : Bool;   // Belebung - SigmaControl Gebläse 1 - Alarme - Externe Meldung 1 Sammelmeldung externe Binärmeldung 1
      BB_G1_KS_AM74 : Bool;   // Belebung - SigmaControl Gebläse 1 - Alarme - Externe Meldung 2 Sammelmeldung externe Binärmeldung 2
      BB_G1_KS_AM75 : Bool;   // Belebung - SigmaControl Gebläse 1 - Alarme - Externe Meldung 3 Sammelmeldung externe Binärmeldung 3
      BB_G1_KS_AM76 : Bool;   // Belebung - SigmaControl Gebläse 1 - Alarme - Schalter p1 freier Schaltpunkt auf Druck p1
      BB_G1_KS_AM77 : Bool;   // Belebung - SigmaControl Gebläse 1 - Alarme - Schalter p2 freier Schaltpunkt auf Druck p2
      BB_G1_KS_AM78 : Bool;   // Belebung - SigmaControl Gebläse 1 - Alarme - Schalter T1 freier Schaltpunkt auf Temperatur T1
      BB_G1_KS_AM79 : Bool;   // Belebung - SigmaControl Gebläse 1 - Alarme - Schalter T2 freier Schaltpunkt auf Temperatur T2
      BB_G1_KS_AM80 : Bool;   // Belebung - SigmaControl Gebläse 1 - Alarme - Schalter Blockdrehzahl freier Schaltpunkt auf Blockdrehzahl
      BB_G1_KS_AM65 : Bool;   // Belebung - SigmaControl Gebläse 1 - Alarme - t3-Sensor-Fehler Fehler Sensor PT100 Öltemperatur
      BB_G1_KS_AM66 : Bool;   // Belebung - SigmaControl Gebläse 1 - Alarme - Reserve
      BB_G1_KS_AM67 : Bool;   // Belebung - SigmaControl Gebläse 1 - Alarme - Reserve
      BB_G1_KS_AM68 : Bool;   // Belebung - SigmaControl Gebläse 1 - Alarme - Reserve
      BB_G1_KS_AM69 : Bool;   // Belebung - SigmaControl Gebläse 1 - Alarme - Reserve
      BB_G1_KS_AM70 : Bool;   // Belebung - SigmaControl Gebläse 1 - Alarme - Schwingungsüberwachung VSE ? Schwingungen an Block oder Motor zu hoch
      BB_G1_KS_AM71 : Bool;   // Belebung - SigmaControl Gebläse 1 - Alarme - Schalter T3
      BB_G1_KS_AM72 : Bool;   // Belebung - SigmaControl Gebläse 1 - Alarme - Schalter T_S
      BB_G1_KS_WM9 : Bool;   // Belebung - SigmaControl Gebläse 1 - Warnungen - Temperatur unter der Schalldämmhaube zu hoch
      BB_G1_KS_WM10 : Bool;   // Belebung - SigmaControl Gebläse 1 - Warnungen - Umgebungstemperatur zu niedrig
      BB_G1_KS_WM11 : Bool;   // Belebung - SigmaControl Gebläse 1 - Warnungen - Differenzdruck zu hoch
      BB_G1_KS_WM12 : Bool;   // Belebung - SigmaControl Gebläse 1 - Warnungen - Differenzdruck zu niedrig
      BB_G1_KS_WM13 : Bool;   // Belebung - SigmaControl Gebläse 1 - Warnungen - Filter verstopft, Verschmutzung des Ansaugfilters
      BB_G1_KS_WM14 : Bool;   // Belebung - SigmaControl Gebläse 1 - Warnungen - Öltemperatur t3 zu hoch
      BB_G1_KS_WM15 : Bool;   // Belebung - SigmaControl Gebläse 1 - Warnungen - Com-Module Kommunikationsfehler Busankopplung über Com-Module ist unterbrochen
      BB_G1_KS_WM16 : Bool;   // Belebung - SigmaControl Gebläse 1 - Warnungen - SAM 4.0 Kommunikationsfehler Busankopplung über Com-Module ist unterbrochen
      BB_G1_KS_WM1 : Bool;   // Belebung - SigmaControl Gebläse 1 - Warnungen - Equipmentnummer unvollständig -> Equipmentnummer des Gebläses hat weniger als sieben Zeichen
      BB_G1_KS_WM2 : Bool;   // Belebung - SigmaControl Gebläse 1 - Warnungen - Sammelwarnung
      BB_G1_KS_WM3 : Bool;   // Belebung - SigmaControl Gebläse 1 - Warnungen - Reserve
      BB_G1_KS_WM4 : Bool;   // Belebung - SigmaControl Gebläse 1 - Warnungen - Schmierölstand Antriebsseite Gebläseblock zu niedrig
      BB_G1_KS_WM5 : Bool;   // Belebung - SigmaControl Gebläse 1 - Warnungen - Schmierölstand Steuerseite Gebläseblock zu niedrig
      BB_G1_KS_WM6 : Bool;   // Belebung - SigmaControl Gebläse 1 - Warnungen - Ansaugtemperatur t1 zu hoch
      BB_G1_KS_WM7 : Bool;   // Belebung - SigmaControl Gebläse 1 - Warnungen - Ansaugtemperatur t1 zu niedrig
      BB_G1_KS_WM8 : Bool;   // Belebung - SigmaControl Gebläse 1 - Warnungen - Verdichtungsendtemperatur t2 zu hoch
      BB_G1_KS_WM25 : Bool;   // Belebung - SigmaControl Gebläse 1 - Warnungen - Motorlager Schaltschrank-Lüfter -> Prüffrist abgelaufen
      BB_G1_KS_WM26 : Bool;   // Belebung - SigmaControl Gebläse 1 - Warnungen - Schmieröl -> Wartungsfrist abgelaufen
      BB_G1_KS_WM27 : Bool;   // Belebung - SigmaControl Gebläse 1 - Warnungen - Reserve
      BB_G1_KS_WM28 : Bool;   // Belebung - SigmaControl Gebläse 1 - Warnungen - Ansaugluftfilter -> Wartungsfrist abgelaufen
      BB_G1_KS_WM29 : Bool;   // Belebung - SigmaControl Gebläse 1 - Warnungen - Filtermatte -> Wartungsfrist abgelaufen
      BB_G1_KS_WM30 : Bool;   // Belebung - SigmaControl Gebläse 1 - Warnungen - Keilriemen -> Wartungsfrist abgelaufen
      BB_G1_KS_WM31 : Bool;   // Belebung - SigmaControl Gebläse 1 - Warnungen - Motorlager -> Wartungsfrist abgelaufen
      BB_G1_KS_WM32 : Bool;   // Belebung - SigmaControl Gebläse 1 - Warnungen - Motorlager Gebläsemotor -> Prüffrist abgelaufen
      BB_G1_KS_WM17 : Bool;   // Belebung - SigmaControl Gebläse 1 - Warnungen - Temperaturdifferenz t2 (VET) - t1 (Ansaugtemperatur) zu hoch
      BB_G1_KS_WM18 : Bool;   // Belebung - SigmaControl Gebläse 1 - Warnungen - Temperatur Gebläsemotor zu hoch
      BB_G1_KS_WM19 : Bool;   // Belebung - SigmaControl Gebläse 1 - Warnungen - Ansaugdruck p1 zu niedrig -> Verschmutzung des Ansaugfilters
      BB_G1_KS_WM20 : Bool;   // Belebung - SigmaControl Gebläse 1 - Warnungen - Enddruck p2 zu hoch
      BB_G1_KS_WM21 : Bool;   // Belebung - SigmaControl Gebläse 1 - Warnungen - Öltemperatur t3 zu niedrig
      BB_G1_KS_WM22 : Bool;   // Belebung - SigmaControl Gebläse 1 - Warnungen - Druckverhältnis über Block zu hoch
      BB_G1_KS_WM23 : Bool;   // Belebung - SigmaControl Gebläse 1 - Warnungen - Reserve
      BB_G1_KS_WM24 : Bool;   // Belebung - SigmaControl Gebläse 1 - Warnungen - maximale Schalthäufigkeit des Netzschützes ist erreicht -> austauschen
      BB_G1_KS_WM41 : Bool;   // Belebung - SigmaControl Gebläse 1 - Warnungen - Reserve
      BB_G1_KS_WM42 : Bool;   // Belebung - SigmaControl Gebläse 1 - Warnungen - Reserve
      BB_G1_KS_WM43 : Bool;   // Belebung - SigmaControl Gebläse 1 - Warnungen - Reserve
      BB_G1_KS_WM44 : Bool;   // Belebung - SigmaControl Gebläse 1 - Warnungen - Reserve
      BB_G1_KS_WM45 : Bool;   // Belebung - SigmaControl Gebläse 1 - Warnungen - Reserve
      BB_G1_KS_WM46 : Bool;   // Belebung - SigmaControl Gebläse 1 - Warnungen - Reserve
      BB_G1_KS_WM47 : Bool;   // Belebung - SigmaControl Gebläse 1 - Warnungen - Elektrobauteile und -installation -> Wartungsfrist abgelaufen
      BB_G1_KS_WM48 : Bool;   // Belebung - SigmaControl Gebläse 1 - Warnungen - Schmierung Motorlager Gebläsemotor -> Wartungsfrist abgelaufen
      BB_G1_KS_WM33 : Bool;   // Belebung - SigmaControl Gebläse 1 - Warnungen - Motorlager Schalldämmhauben-Lüfter -> Prüffrist abgelaufen
      BB_G1_KS_WM34 : Bool;   // Belebung - SigmaControl Gebläse 1 - Warnungen - FU-Lüfter -> Prüffrist abgelaufen
      BB_G1_KS_WM35 : Bool;   // Belebung - SigmaControl Gebläse 1 - Warnungen - Filter Getriebeentlüftung -> Wartungsfrist abgelaufen
      BB_G1_KS_WM36 : Bool;   // Belebung - SigmaControl Gebläse 1 - Warnungen - Maximal zulässige Schalthäufigkeit des Motors in den letzten 60 Minuten überschritten
      BB_G1_KS_WM37 : Bool;   // Belebung - SigmaControl Gebläse 1 - Warnungen - Reserve
      BB_G1_KS_WM38 : Bool;   // Belebung - SigmaControl Gebläse 1 - Warnungen - Ansaugdruck p1 zu niedrig -> Verschmutzung des Ansaugfilters
      BB_G1_KS_WM39 : Bool;   // Belebung - SigmaControl Gebläse 1 - Warnungen - Enddruck p2 zu hoch
      BB_G1_KS_WM40 : Bool;   // Belebung - SigmaControl Gebläse 1 - Warnungen - Überspannung im Stromversorgungsnetz
      BB_G1_KS_WM57 : Bool;   // Belebung - SigmaControl Gebläse 1 - Warnungen - Reserve
      BB_G1_KS_WM58 : Bool;   // Belebung - SigmaControl Gebläse 1 - Warnungen - SC2 zu SC2 Kommunikation unterbrochen
      BB_G1_KS_WM59 : Bool;   // Belebung - SigmaControl Gebläse 1 - Warnungen - Reserve
      BB_G1_KS_WM60 : Bool;   // Belebung - SigmaControl Gebläse 1 - Warnungen - Reserve
      BB_G1_KS_WM61 : Bool;   // Belebung - SigmaControl Gebläse 1 - Warnungen - Reserve
      BB_G1_KS_WM62 : Bool;   // Belebung - SigmaControl Gebläse 1 - Warnungen - FU im Servicebetrieb
      BB_G1_KS_WM63 : Bool;   // Belebung - SigmaControl Gebläse 1 - Warnungen - Test der "Safe Torque off" Abschaltpfade des Frequenzumrichters
      BB_G1_KS_WM64 : Bool;   // Belebung - SigmaControl Gebläse 1 - Warnungen - Reserve
      BB_G1_KS_WM49 : Bool;   // Belebung - SigmaControl Gebläse 1 - Warnungen - Jahreswartung fällig (erscheint 1 Jahr nach letzter Wartung)
      BB_G1_KS_WM50 : Bool;   // Belebung - SigmaControl Gebläse 1 - Warnungen - Fehler beim Schreiben der Daten auf SD-Karte
      BB_G1_KS_WM51 : Bool;   // Belebung - SigmaControl Gebläse 1 - Warnungen - Nachschmiereinrichtung meldet einen Fehler
      BB_G1_KS_WM52 : Bool;   // Belebung - SigmaControl Gebläse 1 - Warnungen - Reserve
      BB_G1_KS_WM53 : Bool;   // Belebung - SigmaControl Gebläse 1 - Warnungen - Reserve
      BB_G1_KS_WM54 : Bool;   // Belebung - SigmaControl Gebläse 1 - Warnungen - Reserve
      BB_G1_KS_WM55 : Bool;   // Belebung - SigmaControl Gebläse 1 - Warnungen - Reserve
      BB_G1_KS_WM56 : Bool;   // Belebung - SigmaControl Gebläse 1 - Warnungen - Reserve
      BB_G1_KS_WM73 : Bool;   // Belebung - SigmaControl Gebläse 1 - Warnungen - Sammelmeldung externe Binärmeldung 1
      BB_G1_KS_WM74 : Bool;   // Belebung - SigmaControl Gebläse 1 - Warnungen - Sammelmeldung externe Binärmeldung 2
      BB_G1_KS_WM75 : Bool;   // Belebung - SigmaControl Gebläse 1 - Warnungen - Sammelmeldung externe Binärmeldung 3
      BB_G1_KS_WM76 : Bool;   // Belebung - SigmaControl Gebläse 1 - Warnungen - Schalter p1 freier Schaltpunkt auf Druck p1
      BB_G1_KS_WM77 : Bool;   // Belebung - SigmaControl Gebläse 1 - Warnungen - Schalter p2 freier Schaltpunkt auf Druck p2
      BB_G1_KS_WM78 : Bool;   // Belebung - SigmaControl Gebläse 1 - Warnungen - Schalter T1 freier Schaltpunkt auf Temperatur T1
      BB_G1_KS_WM79 : Bool;   // Belebung - SigmaControl Gebläse 1 - Warnungen - Schalter T2 freier Schaltpunkt auf Temperatur T2
      BB_G1_KS_WM80 : Bool;   // Belebung - SigmaControl Gebläse 1 - Warnungen - Schalter Blockdrehzahl freier Schaltpunkt auf Blockdrehzahl
      BB_G1_KS_WM65 : Bool;   // Belebung - SigmaControl Gebläse 1 - Warnungen - Reserve
      BB_G1_KS_WM66 : Bool;   // Belebung - SigmaControl Gebläse 1 - Warnungen - Reserve
      BB_G1_KS_WM67 : Bool;   // Belebung - SigmaControl Gebläse 1 - Warnungen - Reserve
      BB_G1_KS_WM68 : Bool;   // Belebung - SigmaControl Gebläse 1 - Warnungen - Schalter T3
      BB_G1_KS_WM69 : Bool;   // Belebung - SigmaControl Gebläse 1 - Warnungen - Schalter T_S
      BB_G1_KS_WM70 : Bool;   // Belebung - SigmaControl Gebläse 1 - Warnungen - Schwingungsüberwachung VSE -> Schwingungen an Block oder Motor
      BB_G1_KS_WM71 : Bool;   // Belebung - SigmaControl Gebläse 1 - Warnungen - Schwingungsüberwachung VSE -> Schwingungen an Block oder Motor
      BB_G1_KS_WM72 : Bool;   // Belebung - SigmaControl Gebläse 1 - Warnungen - Schwingungsüberwachung Summensignal -> Schwingungen an Block oder Motor
      BB_G1_KS_OM9 : Bool;   // Belebung - SigmaControl Gebläse 1 - Betriebsmeldungen - Reserve
      BB_G1_KS_OM10 : Bool;   // Belebung - SigmaControl Gebläse 1 - Betriebsmeldungen - Reserve
      BB_G1_KS_OM11 : Bool;   // Belebung - SigmaControl Gebläse 1 - Betriebsmeldungen - Warten auf Kaltstart -> Temperaturen im Gebläse zu niedrig
      BB_G1_KS_OM12 : Bool;   // Belebung - SigmaControl Gebläse 1 - Betriebsmeldungen - Ölrücklauf vom Filter in die Ölräume gestartet
      BB_G1_KS_OM13 : Bool;   // Belebung - SigmaControl Gebläse 1 - Betriebsmeldungen - Ölmangel (Ölrücklauf abwarten, Ölstand zu niedrig)
      BB_G1_KS_OM14 : Bool;   // Belebung - SigmaControl Gebläse 1 - Betriebsmeldungen - Reserve
      BB_G1_KS_OM15 : Bool;   // Belebung - SigmaControl Gebläse 1 - Betriebsmeldungen - Reserve
      BB_G1_KS_OM16 : Bool;   // Belebung - SigmaControl Gebläse 1 - Betriebsmeldungen - Reserve
      BB_G1_KS_OM1 : Bool;   // Belebung - SigmaControl Gebläse 1 - Betriebsmeldungen - Reserve
      BB_G1_KS_OM2 : Bool;   // Belebung - SigmaControl Gebläse 1 - Betriebsmeldungen - Reserve
      BB_G1_KS_OM3 : Bool;   // Belebung - SigmaControl Gebläse 1 - Betriebsmeldungen - Reserve
      BB_G1_KS_OM4 : Bool;   // Belebung - SigmaControl Gebläse 1 - Betriebsmeldungen - Reserve
      BB_G1_KS_OM5 : Bool;   // Belebung - SigmaControl Gebläse 1 - Betriebsmeldungen - Reserve
      BB_G1_KS_OM6 : Bool;   // Belebung - SigmaControl Gebläse 1 - Betriebsmeldungen - Reserve
      BB_G1_KS_OM7 : Bool;   // Belebung - SigmaControl Gebläse 1 - Betriebsmeldungen - Reserve
      BB_G1_KS_OM8 : Bool;   // Belebung - SigmaControl Gebläse 1 - Betriebsmeldungen - Reserve
      BB_G1_KS_OM25 : Bool;   // Belebung - SigmaControl Gebläse 1 - Betriebsmeldungen - Reserve
      BB_G1_KS_OM26 : Bool;   // Belebung - SigmaControl Gebläse 1 - Betriebsmeldungen - Reserve
      BB_G1_KS_OM27 : Bool;   // Belebung - SigmaControl Gebläse 1 - Betriebsmeldungen - Power OFF -> ON Neustart der Steuerung erforderlich
      BB_G1_KS_OM28 : Bool;   // Belebung - SigmaControl Gebläse 1 - Betriebsmeldungen - Reserve
      BB_G1_KS_OM29 : Bool;   // Belebung - SigmaControl Gebläse 1 - Betriebsmeldungen - Reserve
      BB_G1_KS_OM30 : Bool;   // Belebung - SigmaControl Gebläse 1 - Betriebsmeldungen - Schalter p1 freier Schaltpunkt auf Druck p1
      BB_G1_KS_OM31 : Bool;   // Belebung - SigmaControl Gebläse 1 - Betriebsmeldungen - Schalter p2 freier Schaltpunkt auf Druck p2
      BB_G1_KS_OM32 : Bool;   // Belebung - SigmaControl Gebläse 1 - Betriebsmeldungen - Schalter T1 freier Schaltpunkt auf Temperatur T1
      BB_G1_KS_OM17 : Bool;   // Belebung - SigmaControl Gebläse 1 - Betriebsmeldungen - Externe Meldung 1 Sammelmeldung externe Binärmeldung 1
      BB_G1_KS_OM18 : Bool;   // Belebung - SigmaControl Gebläse 1 - Betriebsmeldungen - Externe Meldung 2 Sammelmeldung externe Binärmeldung 2
      BB_G1_KS_OM19 : Bool;   // Belebung - SigmaControl Gebläse 1 - Betriebsmeldungen - Externe Meldung 3 Sammelmeldung externe Binärmeldung 3
      BB_G1_KS_OM20 : Bool;   // Belebung - SigmaControl Gebläse 1 - Betriebsmeldungen - Schwingungsüberwachung VSE -> Schwingungen an Block oder Motor
      BB_G1_KS_OM21 : Bool;   // Belebung - SigmaControl Gebläse 1 - Betriebsmeldungen - Schwingungsüberwachung Summensignal -> Schwingungen an Block oder Motor
      BB_G1_KS_OM22 : Bool;   // Belebung - SigmaControl Gebläse 1 - Betriebsmeldungen - Reserve
      BB_G1_KS_OM23 : Bool;   // Belebung - SigmaControl Gebläse 1 - Betriebsmeldungen - Reserve
      BB_G1_KS_OM24 : Bool;   // Belebung - SigmaControl Gebläse 1 - Betriebsmeldungen - Reserve
      BB_G1_KS_OM41 : Bool;   // Belebung - SigmaControl Gebläse 1 - Betriebsmeldungen - Reserve
      BB_G1_KS_OM42 : Bool;   // Belebung - SigmaControl Gebläse 1 - Betriebsmeldungen - Reserve
      BB_G1_KS_OM43 : Bool;   // Belebung - SigmaControl Gebläse 1 - Betriebsmeldungen - Reserve
      BB_G1_KS_OM44 : Bool;   // Belebung - SigmaControl Gebläse 1 - Betriebsmeldungen - Reserve
      BB_G1_KS_OM45 : Bool;   // Belebung - SigmaControl Gebläse 1 - Betriebsmeldungen - Reserve
      BB_G1_KS_OM46 : Bool;   // Belebung - SigmaControl Gebläse 1 - Betriebsmeldungen - Reserve
      BB_G1_KS_OM47 : Bool;   // Belebung - SigmaControl Gebläse 1 - Betriebsmeldungen - Reserve
      BB_G1_KS_OM48 : Bool;   // Belebung - SigmaControl Gebläse 1 - Betriebsmeldungen - Reserve
      BB_G1_KS_OM33 : Bool;   // Belebung - SigmaControl Gebläse 1 - Betriebsmeldungen - Schalter T2 freier Schaltpunkt auf Temperatur T2
      BB_G1_KS_OM34 : Bool;   // Belebung - SigmaControl Gebläse 1 - Betriebsmeldungen - Schalter Blockdrehzahl freier Schaltpunkt auf Blockdrehzahl
      BB_G1_KS_OM35 : Bool;   // Belebung - SigmaControl Gebläse 1 - Betriebsmeldungen - Schalter T3
      BB_G1_KS_OM36 : Bool;   // Belebung - SigmaControl Gebläse 1 - Betriebsmeldungen - Schalter T_S
      BB_G1_KS_OM37 : Bool;   // Belebung - SigmaControl Gebläse 1 - Betriebsmeldungen - Reserve
      BB_G1_KS_OM38 : Bool;   // Belebung - SigmaControl Gebläse 1 - Betriebsmeldungen - Ansaugdruck p1 zu niedrig -> Verschmutzung des Ansaugfilters
      BB_G1_KS_OM39 : Bool;   // Belebung - SigmaControl Gebläse 1 - Betriebsmeldungen - Enddruck p2 zu hoch
      BB_G1_KS_OM40 : Bool;   // Belebung - SigmaControl Gebläse 1 - Betriebsmeldungen - Techniker vor Ort Ein Techniker arbeitet an der Maschine
      BB_G1_KS_BS8 : Bool;   // Belebung - SigmaControl Gebläse 1 - Status - Reserve
      BB_G1_KS_BS9 : Bool;   // Belebung - SigmaControl Gebläse 1 - Status - Gebläse Ein (Maschine eingeschaltet)
      BB_G1_KS_BS10 : Bool;   // Belebung - SigmaControl Gebläse 1 - Status - Lüfter Nachkühler Betrieb
      BB_G1_KS_BS11 : Bool;   // Belebung - SigmaControl Gebläse 1 - Status - Lüfter Schalldämmhaube Betrieb
      BB_G1_KS_BS12 : Bool;   // Belebung - SigmaControl Gebläse 1 - Status - Reserve
      BB_G1_KS_BS13 : Bool;   // Belebung - SigmaControl Gebläse 1 - Status - Reserve
      BB_G1_KS_BS14 : Bool;   // Belebung - SigmaControl Gebläse 1 - Status - Sammelwartung
      BB_G1_KS_BS15 : Bool;   // Belebung - SigmaControl Gebläse 1 - Status - Sammelwarnung
      BB_G1_KS_BS0 : Bool;   // Belebung - SigmaControl Gebläse 1 - Status - Anlage Ein + Fernbetrieb Ein + Bus (Receive)
      BB_G1_KS_BS1 : Bool;   // Belebung - SigmaControl Gebläse 1 - Status - Motor Betrieb
      BB_G1_KS_BS2 : Bool;   // Belebung - SigmaControl Gebläse 1 - Status - Lastlauf
      BB_G1_KS_BS3 : Bool;   // Belebung - SigmaControl Gebläse 1 - Status - Leerlauf
      BB_G1_KS_BS4 : Bool;   // Belebung - SigmaControl Gebläse 1 - Status - vor-Ort Betrieb
      BB_G1_KS_BS5 : Bool;   // Belebung - SigmaControl Gebläse 1 - Status - Anlage Ein
      BB_G1_KS_BS6 : Bool;   // Belebung - SigmaControl Gebläse 1 - Status - Sammelstörung
      BB_G1_KS_BS7 : Bool;   // Belebung - SigmaControl Gebläse 1 - Status - Sammelwarnung/-warnung
      BB_G1_KS_BS24 : Bool;   // Belebung - SigmaControl Gebläse 1 - Status - Betriebsart Volumenstromregelung
      BB_G1_KS_BS25 : Bool;   // Belebung - SigmaControl Gebläse 1 - Status - Reserve
      BB_G1_KS_BS26 : Bool;   // Belebung - SigmaControl Gebläse 1 - Status - Reserve
      BB_G1_KS_BS27 : Bool;   // Belebung - SigmaControl Gebläse 1 - Status - Reserve
      BB_G1_KS_BS28 : Bool;   // Belebung - SigmaControl Gebläse 1 - Status - Reserve
      BB_G1_KS_BS29 : Bool;   // Belebung - SigmaControl Gebläse 1 - Status - Reserve
      BB_G1_KS_BS30 : Bool;   // Belebung - SigmaControl Gebläse 1 - Status - Reserve
      BB_G1_KS_BS31 : Bool;   // Belebung - SigmaControl Gebläse 1 - Status - Reserve
      BB_G1_KS_BS16 : Bool;   // Belebung - SigmaControl Gebläse 1 - Status - Modus "Gebläse Ein" nur durch vor-Ort-Bedienung
      BB_G1_KS_BS17 : Bool;   // Belebung - SigmaControl Gebläse 1 - Status - Reserve
      BB_G1_KS_BS18 : Bool;   // Belebung - SigmaControl Gebläse 1 - Status - Reserve
      BB_G1_KS_BS19 : Bool;   // Belebung - SigmaControl Gebläse 1 - Status - Reserve
      BB_G1_KS_BS20 : Bool;   // Belebung - SigmaControl Gebläse 1 - Status - Betriebsart Festdrehzahl
      BB_G1_KS_BS21 : Bool;   // Belebung - SigmaControl Gebläse 1 - Status - Betriebsart externe Drehzahlvorgabe
      BB_G1_KS_BS22 : Bool;   // Belebung - SigmaControl Gebläse 1 - Status - Betriebsart Druckregelung
      BB_G1_KS_BS23 : Bool;   // Belebung - SigmaControl Gebläse 1 - Status - Betriebsart externe Größe
      BB_G1_KS_BS40 : Bool;   // Belebung - SigmaControl Gebläse 1 - Status - Reserve
      BB_G1_KS_BS41 : Bool;   // Belebung - SigmaControl Gebläse 1 - Status - Reserve
      BB_G1_KS_BS42 : Bool;   // Belebung - SigmaControl Gebläse 1 - Status - Reserve
      BB_G1_KS_BS43 : Bool;   // Belebung - SigmaControl Gebläse 1 - Status - Reserve
      BB_G1_KS_BS44 : Bool;   // Belebung - SigmaControl Gebläse 1 - Status - Reserve
      BB_G1_KS_BS45 : Bool;   // Belebung - SigmaControl Gebläse 1 - Status - Reserve
      BB_G1_KS_BS46 : Bool;   // Belebung - SigmaControl Gebläse 1 - Status - Reserve
      BB_G1_KS_BS47 : Bool;   // Belebung - SigmaControl Gebläse 1 - Status - Reserve
      BB_G1_KS_BS32 : Bool;   // Belebung - SigmaControl Gebläse 1 - Status - Reserve
      BB_G1_KS_BS33 : Bool;   // Belebung - SigmaControl Gebläse 1 - Status - Reserve
      BB_G1_KS_BS34 : Bool;   // Belebung - SigmaControl Gebläse 1 - Status - Reserve
      BB_G1_KS_BS35 : Bool;   // Belebung - SigmaControl Gebläse 1 - Status - Reserve
      BB_G1_KS_BS36 : Bool;   // Belebung - SigmaControl Gebläse 1 - Status - Modus Laststeuerung Lastsignal durch ext. Kontakt ist aktiv
      BB_G1_KS_BS37 : Bool;   // Belebung - SigmaControl Gebläse 1 - Status - Reserve
      BB_G1_KS_BS38 : Bool;   // Belebung - SigmaControl Gebläse 1 - Status - Modus Laststeuerung Lastsignal durch BusMaster ist aktiv
      BB_G1_KS_BS39 : Bool;   // Belebung - SigmaControl Gebläse 1 - Status - Reserve
      BB_G1_KS_BS56 : Bool;   // Belebung - SigmaControl Gebläse 1 - Status - Reserve
      BB_G1_KS_BS57 : Bool;   // Belebung - SigmaControl Gebläse 1 - Status - Reserve
      BB_G1_KS_BS58 : Bool;   // Belebung - SigmaControl Gebläse 1 - Status - Reserve
      BB_G1_KS_BS59 : Bool;   // Belebung - SigmaControl Gebläse 1 - Status - Reserve
      BB_G1_KS_BS60 : Bool;   // Belebung - SigmaControl Gebläse 1 - Status - Reserve
      BB_G1_KS_BS61 : Bool;   // Belebung - SigmaControl Gebläse 1 - Status - Reserve
      BB_G1_KS_BS62 : Bool;   // Belebung - SigmaControl Gebläse 1 - Status - Reserve
      BB_G1_KS_BS63 : Bool;   // Belebung - SigmaControl Gebläse 1 - Status - Reserve
      BB_G1_KS_BS48 : Bool;   // Belebung - SigmaControl Gebläse 1 - Status - Reserve
      BB_G1_KS_BS49 : Bool;   // Belebung - SigmaControl Gebläse 1 - Status - Reserve
      BB_G1_KS_BS50 : Bool;   // Belebung - SigmaControl Gebläse 1 - Status - Reserve
      BB_G1_KS_BS51 : Bool;   // Belebung - SigmaControl Gebläse 1 - Status - Automatischer Anlauf nach Netzspannung EIN
      BB_G1_KS_BS52 : Bool;   // Belebung - SigmaControl Gebläse 1 - Status - Reserve
      BB_G1_KS_BS53 : Bool;   // Belebung - SigmaControl Gebläse 1 - Status - Reserve
      BB_G1_KS_BS54 : Bool;   // Belebung - SigmaControl Gebläse 1 - Status - Reserve
      BB_G1_KS_BS55 : Bool;   // Belebung - SigmaControl Gebläse 1 - Status - Meldungs-Quittierung durch Master
      BB_G2_KS_AM9 : Bool;   // Belebung - SigmaControl Gebläse 2 - Alarme - Zulässige Innentemperatur von SIGMA CONTROL 2 MCS oder IOM überschritten
      BB_G2_KS_AM10 : Bool;   // Belebung - SigmaControl Gebläse 2 - Alarme - Enddruck p2 zu hoch
      BB_G2_KS_AM11 : Bool;   // Belebung - SigmaControl Gebläse 2 - Alarme - Reserve
      BB_G2_KS_AM12 : Bool;   // Belebung - SigmaControl Gebläse 2 - Alarme - Reserve
      BB_G2_KS_AM13 : Bool;   // Belebung - SigmaControl Gebläse 2 - Alarme - Überlast Gebläsemotor -> Abschaltung wegen Überlastung
      BB_G2_KS_AM14 : Bool;   // Belebung - SigmaControl Gebläse 2 - Alarme - Abschaltung des Nachkühler-Lüfters wegen Überlastung
      BB_G2_KS_AM15 : Bool;   // Belebung - SigmaControl Gebläse 2 - Alarme - Maximal zulässige Verdichtungs-Endtemperatur (VET) überschritten
      BB_G2_KS_AM16 : Bool;   // Belebung - SigmaControl Gebläse 2 - Alarme - Reserve
      BB_G2_KS_AM1 : Bool;   // Belebung - SigmaControl Gebläse 2 - Alarme - Reserve
      BB_G2_KS_AM2 : Bool;   // Belebung - SigmaControl Gebläse 2 - Alarme - Temperatur Gebläsemotor zu hoch
      BB_G2_KS_AM3 : Bool;   // Belebung - SigmaControl Gebläse 2 - Alarme - Reserve
      BB_G2_KS_AM4 : Bool;   // Belebung - SigmaControl Gebläse 2 - Alarme - NOT-HALT-Befehlsgerät betätigt
      BB_G2_KS_AM5 : Bool;   // Belebung - SigmaControl Gebläse 2 - Alarme - Schmierölstand Antriebsseite Gebläseblock zu niedrig
      BB_G2_KS_AM6 : Bool;   // Belebung - SigmaControl Gebläse 2 - Alarme - Schmierölstand Steuerseite Gebläseblock zu niedrig
      BB_G2_KS_AM7 : Bool;   // Belebung - SigmaControl Gebläse 2 - Alarme - Phasenfehler oder Unter-/Überspannung Gebläsemotor
      BB_G2_KS_AM8 : Bool;   // Belebung - SigmaControl Gebläse 2 - Alarme - Diagnose-Sammelmeldung
      BB_G2_KS_AM25 : Bool;   // Belebung - SigmaControl Gebläse 2 - Alarme - Sammelfehler IOM
      BB_G2_KS_AM26 : Bool;   // Belebung - SigmaControl Gebläse 2 - Alarme - Reserve
      BB_G2_KS_AM27 : Bool;   // Belebung - SigmaControl Gebläse 2 - Alarme - Filter verstopft -> Verschmutzung des Ansaugfilters
      BB_G2_KS_AM28 : Bool;   // Belebung - SigmaControl Gebläse 2 - Alarme - Öltemperatur t3 sehr hoch
      BB_G2_KS_AM29 : Bool;   // Belebung - SigmaControl Gebläse 2 - Alarme - Reserve
      BB_G2_KS_AM30 : Bool;   // Belebung - SigmaControl Gebläse 2 - Alarme - Reserve
      BB_G2_KS_AM31 : Bool;   // Belebung - SigmaControl Gebläse 2 - Alarme - Temperaturdifferenz t2 (VET) - t1 (Ansaugtemperatur) zu hoch
      BB_G2_KS_AM32 : Bool;   // Belebung - SigmaControl Gebläse 2 - Alarme - Druckverhältnis über Block zu hoch
      BB_G2_KS_AM17 : Bool;   // Belebung - SigmaControl Gebläse 2 - Alarme - Reserve
      BB_G2_KS_AM18 : Bool;   // Belebung - SigmaControl Gebläse 2 - Alarme - Abschaltung des Schalldämmhauben-Lüfters wegen Überlastung
